(* IEC 61131-3 sources: mect_apps/AnyTPAC/TestSuite/plc (part 2) *)

(* ---- eq_P.st ---- *)
(*[[
]]*)
PROGRAM eq_P
#import "Crosstable.gvl"
#import "Resource1.gvl"
CONST
	this : int := 36;
	test_cases : int := 6;
END_CONST
VAR
	test_case : array [1..test_cases] of any2_bool_T := [
		(input0 :=  10.0, input1 :=  10.0, retval := true),
		(input0 :=  10.0, input1 :=  20.0, retval := false),
		(input0 :=  10.0, input1 :=  5.0,  retval := false),
		(input0 :=  -100.0, input1 := -100.0,  retval := true),
		(input0 :=  -100.0, input1 := 7.0,  retval := false),
		(input0 :=  -100.0, input1 := 109.0,  retval := false)
	];
	ret_bool   : bool;
	ret_byte   : bool;
	ret_dint   : bool;
	ret_dword  : bool;
	ret_int    : bool;
	ret_lreal  : bool;
	ret_real   : bool;
	ret_string : bool;
	ret_time   : bool;
	ret_uint   : bool;
	ret_udint  : bool;
	ret_word   : bool;

	expected_ret_bool   : bool;
	expected_ret_byte   : bool;
	expected_ret_dint   : bool;
	expected_ret_dword  : bool;
	expected_ret_int    : bool;
	expected_ret_lreal  : bool;
	expected_ret_real   : bool;
	expected_ret_string : bool;
	expected_ret_time   : bool;
	expected_ret_uint   : bool;
	expected_ret_udint  : bool;
	expected_ret_word   : bool;

	index : int := 1;
	expected: string;
	obtained: string;
	result : bool;
END_VAR

	if Status = STATUS_RUNNING AND test_level_36 > TEST_DISABLED and test_loops_36 < Target then

		(* ---------- test action ---------------*)
        ret_bool   := eq( lreal_to_bool(test_case[index].input0),
						 lreal_to_bool(test_case[index].input1));
        ret_byte   := eq( lreal_to_byte(test_case[index].input0),
						 lreal_to_byte(test_case[index].input1));
        ret_dint   := eq( lreal_to_dint(test_case[index].input0),
						 lreal_to_dint(test_case[index].input1));
        ret_dword  := eq( lreal_to_dword(test_case[index].input0),
						 lreal_to_dword(test_case[index].input1));
        ret_int    := eq( lreal_to_int(test_case[index].input0),
						 lreal_to_int(test_case[index].input1));
        ret_lreal  := eq( test_case[index].input0,
						 test_case[index].input1);
        ret_real   := eq( lreal_to_real(test_case[index].input0),
						 lreal_to_real(test_case[index].input1));
        ret_string := eq(lreal_to_string(test_case[index].input0),
						 lreal_to_string(test_case[index].input1));
        ret_time   := eq( lreal_to_time(test_case[index].input0),
						 lreal_to_time(test_case[index].input1));
        ret_uint   := eq( lreal_to_uint(test_case[index].input0),
						 lreal_to_uint(test_case[index].input1));
        ret_udint  := eq(lreal_to_udint(test_case[index].input0),
						 lreal_to_udint(test_case[index].input1));
        ret_word   := eq( lreal_to_word(test_case[index].input0),
						 lreal_to_word(test_case[index].input1));

		IF (test_case[index].input0 <> 0.0 and test_case[index].input1 <> 0.0)
			or (test_case[index].input0 = 0.0 and test_case[index].input1 = 0.0)THEN
        	expected_ret_bool   := true;
        ELSE
        	expected_ret_bool   := false;
		END_IF;

		expected_ret_byte   := test_case[index].retval;
		expected_ret_dint   := test_case[index].retval;
		expected_ret_dword  := test_case[index].retval;
		expected_ret_int    := test_case[index].retval;
		expected_ret_lreal  := test_case[index].retval;
		expected_ret_real   := test_case[index].retval;
		expected_ret_string := test_case[index].retval;
		expected_ret_time   := test_case[index].retval;
		expected_ret_uint   := test_case[index].retval;
		expected_ret_udint  := test_case[index].retval;
		expected_ret_word   := test_case[index].retval;

		(* ---------- test condition ---------------*)
        result := (ret_bool = expected_ret_bool)
				  and (ret_byte = expected_ret_byte)
				  and (ret_dint = expected_ret_dint)
				  and (ret_dword = expected_ret_dword)
				  and (ret_int = expected_ret_int)
				  and (ret_lreal = expected_ret_lreal)
				  and (ret_real = expected_ret_real)
				  and (ret_string = expected_ret_string)
				  and (ret_time = expected_ret_time)
				  and (ret_uint = expected_ret_uint)
				  and (ret_udint = expected_ret_udint)
				  and (ret_word = expected_ret_word);

		(* ---------- log message ---------------*)
		expected := '';
		expected := CONCAT(expected, comma_blank, bool_to_string(expected_ret_bool));
		expected := CONCAT(expected, comma_blank, bool_to_string(expected_ret_byte));
		expected := CONCAT(expected, comma_blank, bool_to_string(expected_ret_dint));
		expected := CONCAT(expected, comma_blank, bool_to_string(expected_ret_dword));
		expected := CONCAT(expected, comma_blank, bool_to_string(expected_ret_int));
		expected := CONCAT(expected, comma_blank, bool_to_string(expected_ret_lreal));
		expected := CONCAT(expected, comma_blank, bool_to_string(expected_ret_real));
		expected := CONCAT(expected, comma_blank, bool_to_string(expected_ret_string));
		expected := CONCAT(expected, comma_blank, bool_to_string(expected_ret_time));
		expected := CONCAT(expected, comma_blank, bool_to_string(expected_ret_uint));
		expected := CONCAT(expected, comma_blank, bool_to_string(expected_ret_udint));
		expected := CONCAT(expected, comma_blank, bool_to_string(expected_ret_word));

		obtained := '';
		obtained := CONCAT(obtained, comma_blank, bool_to_string(ret_bool));
		obtained := CONCAT(obtained, comma_blank, bool_to_string(ret_byte));
		obtained := CONCAT(obtained, comma_blank, bool_to_string(ret_dint));
		obtained := CONCAT(obtained, comma_blank, bool_to_string(ret_dword));
		obtained := CONCAT(obtained, comma_blank, bool_to_string(ret_int));
		obtained := CONCAT(obtained, comma_blank, bool_to_string(ret_lreal));
		obtained := CONCAT(obtained, comma_blank, bool_to_string(ret_real));
		obtained := CONCAT(obtained, comma_blank, bool_to_string(ret_string));
		obtained := CONCAT(obtained, comma_blank, bool_to_string(ret_time));
		obtained := CONCAT(obtained, comma_blank, bool_to_string(ret_uint));
		obtained := CONCAT(obtained, comma_blank, bool_to_string(ret_udint));
		obtained := CONCAT(obtained, comma_blank, bool_to_string(ret_word));

		(* ---------- cycle ----------*)
		SingleTest(this, result, expected, obtained, test_cases,
				   index, test_level_36, test_counter_36, test_loops_36, test_errors_36);
	end_if;

END_PROGRAM

(* ---- expt_P.st ---- *)
(*[[ ]]*)
PROGRAM expt_P
#import "Crosstable.gvl"
#import "Resource1.gvl"
CONST
	this : int := 20;
	test_cases : int := 5;
	xl : lreal := 0.0000000000001;
	x : real := 0.0000000000001;
END_CONST
VAR
	test_case : array [1..test_cases] of num2_num_T := [
		(input0 := 2.0, input1 := 2.0, ret_real := 4.0, ret_lreal := 4.0),
		(input0 := 2.0, input1 := 3.0, ret_real := 8.0, ret_lreal := 8.0),
		(input0 := 10.0, input1 := 2.0, ret_real := 100.0, ret_lreal := 100.0),
		(input0 := 5.0, input1 := 3.0, ret_real := 125.0, ret_lreal := 125.0),
		(input0 := 10.0, input1 := -1.0, ret_real := 0.1, ret_lreal := 0.1)
	];
    ret_real_int    : real;
    ret_real_dint   : real;
    ret_real_real   : real;
    ret_real_lreal  : real;
    ret_lreal_int   : lreal;
    ret_lreal_dint  : lreal;
    ret_lreal_real  : lreal;
    ret_lreal_lreal : lreal;

	index : int := 1;
	expected : string;
	obtained : string;
	result : bool;
END_VAR

	if Status = STATUS_RUNNING AND test_level_20 > TEST_DISABLED and test_loops_20 < Target then

		(* ---------- test action ---------------*)
        ret_real_int   := expt(lreal_to_real(test_case[index].input0), lreal_to_int(test_case[index].input1));
        ret_real_dint  := expt(lreal_to_real(test_case[index].input0), lreal_to_dint(test_case[index].input1));
        ret_real_real  := expt(lreal_to_real(test_case[index].input0), lreal_to_real(test_case[index].input1));
        ret_real_lreal := expt(lreal_to_real(test_case[index].input0), test_case[index].input1);

        ret_lreal_int   := expt(test_case[index].input0, lreal_to_int(test_case[index].input1));
        ret_lreal_dint  := expt(test_case[index].input0, lreal_to_dint(test_case[index].input1));
        ret_lreal_real  := expt(test_case[index].input0, lreal_to_real(test_case[index].input1));
        ret_lreal_lreal := expt(test_case[index].input0, test_case[index].input1);

		(* ---------- test condition ---------------*)
        result := ((abs(ret_real_int - test_case[index].ret_real) < x)
		      and (abs(ret_real_dint - test_case[index].ret_real) < x)
		      and (abs(ret_real_real - test_case[index].ret_real) < x)
		      and (abs(ret_real_lreal - test_case[index].ret_real) < x)
			  and (abs(ret_lreal_int - test_case[index].ret_lreal) < xl)
		      and (abs(ret_lreal_dint - test_case[index].ret_lreal) < xl)
		      and (abs(ret_lreal_real - test_case[index].ret_lreal) < xl)
		      and (abs(ret_lreal_lreal - test_case[index].ret_lreal) < xl));

		(* ---------- log message ---------------*)
		expected := '';
		expected := CONCAT(expected, comma_blank, real_to_string(test_case[index].ret_real));
		expected := CONCAT(expected, comma_blank, real_to_string(test_case[index].ret_real));
		expected := CONCAT(expected, comma_blank, real_to_string(test_case[index].ret_real));
		expected := CONCAT(expected, comma_blank, real_to_string(test_case[index].ret_real));
		expected := CONCAT(expected, comma_blank, lreal_to_string(test_case[index].ret_lreal));
		expected := CONCAT(expected, comma_blank, lreal_to_string(test_case[index].ret_lreal));
		expected := CONCAT(expected, comma_blank, lreal_to_string(test_case[index].ret_lreal));
		expected := CONCAT(expected, comma_blank, lreal_to_string(test_case[index].ret_lreal));
		obtained := '';
		obtained := CONCAT(obtained, comma_blank, real_to_string(ret_real_int));
		obtained := CONCAT(obtained, comma_blank, real_to_string(ret_real_dint));
		obtained := CONCAT(obtained, comma_blank, real_to_string(ret_real_real));
		obtained := CONCAT(obtained, comma_blank, real_to_string(ret_real_lreal));
		obtained := CONCAT(obtained, comma_blank, lreal_to_string(ret_lreal_int));
		obtained := CONCAT(obtained, comma_blank, lreal_to_string(ret_lreal_dint));
		obtained := CONCAT(obtained, comma_blank, lreal_to_string(ret_lreal_real));
		obtained := CONCAT(obtained, comma_blank, lreal_to_string(ret_lreal_lreal));

		(* ---------- cycle ----------*)
		SingleTest(this, result, expected, obtained, test_cases,
				   index, test_level_20, test_counter_20, test_loops_20, test_errors_20);
	end_if;
END_PROGRAM

(* ---- f_r_trig_P.st ---- *)
(*[[
]]*)
PROGRAM f_r_trig_P
#import "Crosstable.gvl"
#import "Resource1.gvl"
CONST
	this : int := 53;
	test_cases : int := 5;
END_CONST
VAR
	test_case : array [1..test_cases] of bool_bool2_T := [
		(input := false, retval1 := false, retval2 := false),
		(input := true,  retval1 := false, retval2 := true ),
		(input := true,  retval1 := false, retval2 := false),
		(input := false, retval1 := true,  retval2 := false),
		(input := false, retval1 := false, retval2 := false)
	];
    retval1  : bool;
    retval2  : bool;

	F_TRIG_Inst : f_trig;
	R_TRIG_Inst : r_trig;
	index : int := 1;
	expected : string;
	obtained : string;
	result : bool;
END_VAR

	if Status = STATUS_RUNNING AND test_level_53 > TEST_DISABLED and test_loops_53 < Target then

		(* ---------- test action ---------------*)
		F_TRIG_Inst(CLK := test_case[index].input, Q => retval1);
		R_TRIG_Inst(CLK := test_case[index].input, Q => retval2);

		(* ---------- test condition ---------------*)
        result := (retval1 = test_case[index].retval1)
		      and (retval2 = test_case[index].retval2);

		(* ---------- log message ---------------*)
		expected := '';
		expected := CONCAT(expected, comma_blank, bool_to_string(test_case[index].retval1));
		expected := CONCAT(expected, comma_blank, bool_to_string(test_case[index].retval2));
		obtained := '';
		obtained := CONCAT(obtained, comma_blank, bool_to_string(retval1));
		obtained := CONCAT(obtained, comma_blank, bool_to_string(retval2));

		(* ---------- cycle ----------*)
		SingleTest(this, result, expected, obtained, test_cases,
				   index, test_level_53, test_counter_53, test_loops_53, test_errors_53);
	end_if;
END_PROGRAM

(* ---- find_P.st ---- *)
(*[[ ]]*)
PROGRAM find_P
#import "Crosstable.gvl"
#import "Resource1.gvl"
CONST
	this : int := 44;
	test_cases : int := 4;
END_CONST
VAR
	test_case : array [1..test_cases] of string2_int_T := [
		(input0 := 'stringa_in_cui_eseguire_la_ricerca', input1 := 'stringa',  retval := 1),
		(input0 := 'stringa_in_cui_eseguire_la_ricerca', input1 := 'in_cui',   retval := 9),
		(input0 := 'stringa_in_cui_eseguire_la_ricerca', input1 := 'ricerca',  retval := 28),
		(input0 := 'stringa_in_cui_eseguire_la_ricerca', input1 := 'stringa_che_non_esiste',  retval := 0)
	];
    retval0   : int;
    retval1   : dint;

	index : int := 1;
	expected : string;
	obtained : string;
	result : bool;
END_VAR

	if Status = STATUS_RUNNING AND test_level_44 > TEST_DISABLED and test_loops_44 < Target then

		(* ---------- test action ---------------*)
        retval0 := find(test_case[index].input0, test_case[index].input1);
        retval1 := find(test_case[index].input0, test_case[index].input1);

		(* ---------- test condition ---------------*)
        result := (retval0 = test_case[index].retval)
		      and (retval1 = int_to_dint(test_case[index].retval));

		(* ---------- log message ---------------*)
		expected := '';
		expected := CONCAT(expected, comma_blank, int_to_string(test_case[index].retval));
		expected := CONCAT(expected, comma_blank, int_to_string(test_case[index].retval));
		obtained := '';
		obtained := CONCAT(obtained, comma_blank, int_to_string(retval0));
		obtained := CONCAT(obtained, comma_blank, dint_to_string(retval1));

		(* ---------- cycle ----------*)
		SingleTest(this, result, expected, obtained, test_cases,
				   index, test_level_44, test_counter_44, test_loops_44, test_errors_44);
	end_if;
END_PROGRAM

(* ---- ge_P.st ---- *)
(*[[
]]*)
PROGRAM ge_P
#import "Crosstable.gvl"
#import "Resource1.gvl"
CONST
	this : int := 37;
	test_cases : int := 4;
END_CONST
VAR
	test_case : array [1..test_cases] of any2_bool_T := [
		(input0 :=  10.0, input1 :=  10.0, retval := true),
		(input0 :=  10.0, input1 :=  20.0, retval := false),
		(input0 :=  20.0, input1 :=  10.0,  retval := true),
		(input0 :=  -100.0, input1 := -100.0,  retval := true)
	];
	ret_bool   : bool;
	ret_byte   : bool;
	ret_dint   : bool;
	ret_dword  : bool;
	ret_int    : bool;
	ret_lreal  : bool;
	ret_real   : bool;
	ret_string : bool;
	ret_time   : bool;
	ret_uint   : bool;
	ret_udint  : bool;
	ret_word   : bool;

	expected_ret_bool   : bool;
	expected_ret_byte   : bool;
	expected_ret_dint   : bool;
	expected_ret_dword  : bool;
	expected_ret_int    : bool;
	expected_ret_lreal  : bool;
	expected_ret_real   : bool;
	expected_ret_string : bool;
	expected_ret_time   : bool;
	expected_ret_uint   : bool;
	expected_ret_udint  : bool;
	expected_ret_word   : bool;

	index : int := 1;
	expected: string;
	obtained: string;
	result : bool;
END_VAR

	if Status = STATUS_RUNNING AND test_level_37 > TEST_DISABLED and test_loops_37 < Target then

		(* ---------- test action ---------------*)
        ret_bool   := ge( lreal_to_bool(test_case[index].input0),
						 lreal_to_bool(test_case[index].input1));
        ret_byte   := ge( lreal_to_byte(test_case[index].input0),
						 lreal_to_byte(test_case[index].input1));
        ret_dint   := ge( lreal_to_dint(test_case[index].input0),
						 lreal_to_dint(test_case[index].input1));
        ret_dword  := ge( lreal_to_dword(test_case[index].input0),
						 lreal_to_dword(test_case[index].input1));
        ret_int    := ge( lreal_to_int(test_case[index].input0),
						 lreal_to_int(test_case[index].input1));
        ret_lreal  := ge( test_case[index].input0,
						 test_case[index].input1);
        ret_real   := ge( lreal_to_real(test_case[index].input0),
						 lreal_to_real(test_case[index].input1));
        ret_string := ge(lreal_to_string(test_case[index].input0),
						 lreal_to_string(test_case[index].input1));
        ret_time   := ge( lreal_to_time(test_case[index].input0),
						 lreal_to_time(test_case[index].input1));
        ret_uint   := ge( lreal_to_uint(test_case[index].input0),
						 lreal_to_uint(test_case[index].input1));
        ret_udint  := ge(lreal_to_udint(test_case[index].input0),
						 lreal_to_udint(test_case[index].input1));
        ret_word   := ge( lreal_to_word(test_case[index].input0),
						 lreal_to_word(test_case[index].input1));

		IF (test_case[index].input0 <> 0.0 and test_case[index].input1 <> 0.0)
			or (test_case[index].input0 = 0.0 and test_case[index].input1 = 0.0)THEN
        	expected_ret_bool   := true;
        ELSE
        	expected_ret_bool   := false;
		END_IF;
		expected_ret_byte   := test_case[index].retval;
		expected_ret_dint   := test_case[index].retval;
		expected_ret_dword  := test_case[index].retval;
		expected_ret_int    := test_case[index].retval;
		expected_ret_lreal  := test_case[index].retval;
		expected_ret_real   := test_case[index].retval;
		expected_ret_string := test_case[index].retval;
		expected_ret_time   := test_case[index].retval;
		expected_ret_uint   := test_case[index].retval;
		expected_ret_udint  := test_case[index].retval;
		expected_ret_word   := test_case[index].retval;

		(* ---------- test condition ---------------*)
        result := (ret_bool = expected_ret_bool)
				  and (ret_byte = expected_ret_byte)
				  and (ret_dint = expected_ret_dint)
				  and (ret_dword = expected_ret_dword)
				  and (ret_int = expected_ret_int)
				  and (ret_lreal = expected_ret_lreal)
				  and (ret_real = expected_ret_real)
				  and (ret_string = expected_ret_string)
				  and (ret_time = expected_ret_time)
				  and (ret_uint = expected_ret_uint)
				  and (ret_udint = expected_ret_udint)
				  and (ret_word = expected_ret_word);

		(* ---------- log message ---------------*)
		expected := '';
		expected := CONCAT(expected, comma_blank, bool_to_string(expected_ret_bool));
		expected := CONCAT(expected, comma_blank, bool_to_string(expected_ret_byte));
		expected := CONCAT(expected, comma_blank, bool_to_string(expected_ret_dint));
		expected := CONCAT(expected, comma_blank, bool_to_string(expected_ret_dword));
		expected := CONCAT(expected, comma_blank, bool_to_string(expected_ret_int));
		expected := CONCAT(expected, comma_blank, bool_to_string(expected_ret_lreal));
		expected := CONCAT(expected, comma_blank, bool_to_string(expected_ret_real));
		expected := CONCAT(expected, comma_blank, bool_to_string(expected_ret_string));
		expected := CONCAT(expected, comma_blank, bool_to_string(expected_ret_time));
		expected := CONCAT(expected, comma_blank, bool_to_string(expected_ret_uint));
		expected := CONCAT(expected, comma_blank, bool_to_string(expected_ret_udint));
		expected := CONCAT(expected, comma_blank, bool_to_string(expected_ret_word));

		obtained := '';
		obtained := CONCAT(obtained, comma_blank, bool_to_string(ret_bool));
		obtained := CONCAT(obtained, comma_blank, bool_to_string(ret_byte));
		obtained := CONCAT(obtained, comma_blank, bool_to_string(ret_dint));
		obtained := CONCAT(obtained, comma_blank, bool_to_string(ret_dword));
		obtained := CONCAT(obtained, comma_blank, bool_to_string(ret_int));
		obtained := CONCAT(obtained, comma_blank, bool_to_string(ret_lreal));
		obtained := CONCAT(obtained, comma_blank, bool_to_string(ret_real));
		obtained := CONCAT(obtained, comma_blank, bool_to_string(ret_string));
		obtained := CONCAT(obtained, comma_blank, bool_to_string(ret_time));
		obtained := CONCAT(obtained, comma_blank, bool_to_string(ret_uint));
		obtained := CONCAT(obtained, comma_blank, bool_to_string(ret_udint));
		obtained := CONCAT(obtained, comma_blank, bool_to_string(ret_word));

		(* ---------- cycle ----------*)
		SingleTest(this, result, expected, obtained, test_cases,
				   index, test_level_37, test_counter_37, test_loops_37, test_errors_37);
	end_if;

END_PROGRAM

(* ---- gt_P.st ---- *)
(*[[
]]*)
PROGRAM gt_P
#import "Crosstable.gvl"
#import "Resource1.gvl"
CONST
	this : int := 38;
	test_cases : int := 4;
END_CONST
VAR
	test_case : array [1..test_cases] of any2_bool_T := [
		(input0 :=  10.0, input1 :=  10.0, retval := false),
		(input0 :=  10.0, input1 :=  20.0, retval := false),
		(input0 :=  20.0, input1 :=  10.0,  retval := true),
		(input0 :=  -100.0, input1 := -100.0,  retval := false)
	];
	ret_bool   : bool;
	ret_byte   : bool;
	ret_dint   : bool;
	ret_dword  : bool;
	ret_int    : bool;
	ret_lreal  : bool;
	ret_real   : bool;
	ret_string : bool;
	ret_time   : bool;
	ret_uint   : bool;
	ret_udint  : bool;
	ret_word   : bool;

	expected_ret_bool   : bool;
	expected_ret_byte   : bool;
	expected_ret_dint   : bool;
	expected_ret_dword  : bool;
	expected_ret_int    : bool;
	expected_ret_lreal  : bool;
	expected_ret_real   : bool;
	expected_ret_string : bool;
	expected_ret_time   : bool;
	expected_ret_uint   : bool;
	expected_ret_udint  : bool;
	expected_ret_word   : bool;

	index : int := 1;
	expected: string;
	obtained: string;
	result : bool;
END_VAR

	if Status = STATUS_RUNNING AND test_level_38 > TEST_DISABLED and test_loops_38 < Target then

		(* ---------- test action ---------------*)
        ret_bool   := gt( lreal_to_bool(test_case[index].input0),
						 lreal_to_bool(test_case[index].input1));
        ret_byte   := gt( lreal_to_byte(test_case[index].input0),
						 lreal_to_byte(test_case[index].input1));
        ret_dint   := gt( lreal_to_dint(test_case[index].input0),
						 lreal_to_dint(test_case[index].input1));
        ret_dword  := gt( lreal_to_dword(test_case[index].input0),
						 lreal_to_dword(test_case[index].input1));
        ret_int    := gt( lreal_to_int(test_case[index].input0),
						 lreal_to_int(test_case[index].input1));
        ret_lreal  := gt( test_case[index].input0,
						 test_case[index].input1);
        ret_real   := gt( lreal_to_real(test_case[index].input0),
						 lreal_to_real(test_case[index].input1));
        ret_string := gt(lreal_to_string(test_case[index].input0),
						 lreal_to_string(test_case[index].input1));
        ret_time   := gt( lreal_to_time(test_case[index].input0),
						 lreal_to_time(test_case[index].input1));
        ret_uint   := gt( lreal_to_uint(test_case[index].input0),
						 lreal_to_uint(test_case[index].input1));
        ret_udint  := gt(lreal_to_udint(test_case[index].input0),
						 lreal_to_udint(test_case[index].input1));
        ret_word   := gt( lreal_to_word(test_case[index].input0),
						 lreal_to_word(test_case[index].input1));

		IF (test_case[index].input0 <> 0.0 and test_case[index].input1 <> 0.0)
			or (test_case[index].input0 = 0.0 and test_case[index].input1 = 0.0)THEN
        	expected_ret_bool   := false;
        ELSE
        	expected_ret_bool   := true;
		END_IF;
		expected_ret_byte   := test_case[index].retval;
		expected_ret_dint   := test_case[index].retval;
		expected_ret_dword  := test_case[index].retval;
		expected_ret_int    := test_case[index].retval;
		expected_ret_lreal  := test_case[index].retval;
		expected_ret_real   := test_case[index].retval;
		expected_ret_string := test_case[index].retval;
		expected_ret_time   := test_case[index].retval;
		expected_ret_uint   := test_case[index].retval;
		expected_ret_udint  := test_case[index].retval;
		expected_ret_word   := test_case[index].retval;

		(* ---------- test condition ---------------*)
        result := (ret_bool = expected_ret_bool)
				  and (ret_byte = expected_ret_byte)
				  and (ret_dint = expected_ret_dint)
				  and (ret_dword = expected_ret_dword)
				  and (ret_int = expected_ret_int)
				  and (ret_lreal = expected_ret_lreal)
				  and (ret_real = expected_ret_real)
				  and (ret_string = expected_ret_string)
				  and (ret_time = expected_ret_time)
				  and (ret_uint = expected_ret_uint)
				  and (ret_udint = expected_ret_udint)
				  and (ret_word = expected_ret_word);

		(* ---------- log message ---------------*)
		expected := '';
		expected := CONCAT(expected, comma_blank, bool_to_string(expected_ret_bool));
		expected := CONCAT(expected, comma_blank, bool_to_string(expected_ret_byte));
		expected := CONCAT(expected, comma_blank, bool_to_string(expected_ret_dint));
		expected := CONCAT(expected, comma_blank, bool_to_string(expected_ret_dword));
		expected := CONCAT(expected, comma_blank, bool_to_string(expected_ret_int));
		expected := CONCAT(expected, comma_blank, bool_to_string(expected_ret_lreal));
		expected := CONCAT(expected, comma_blank, bool_to_string(expected_ret_real));
		expected := CONCAT(expected, comma_blank, bool_to_string(expected_ret_string));
		expected := CONCAT(expected, comma_blank, bool_to_string(expected_ret_time));
		expected := CONCAT(expected, comma_blank, bool_to_string(expected_ret_uint));
		expected := CONCAT(expected, comma_blank, bool_to_string(expected_ret_udint));
		expected := CONCAT(expected, comma_blank, bool_to_string(expected_ret_word));

		obtained := '';
		obtained := CONCAT(obtained, comma_blank, bool_to_string(ret_bool));
		obtained := CONCAT(obtained, comma_blank, bool_to_string(ret_byte));
		obtained := CONCAT(obtained, comma_blank, bool_to_string(ret_dint));
		obtained := CONCAT(obtained, comma_blank, bool_to_string(ret_dword));
		obtained := CONCAT(obtained, comma_blank, bool_to_string(ret_int));
		obtained := CONCAT(obtained, comma_blank, bool_to_string(ret_lreal));
		obtained := CONCAT(obtained, comma_blank, bool_to_string(ret_real));
		obtained := CONCAT(obtained, comma_blank, bool_to_string(ret_string));
		obtained := CONCAT(obtained, comma_blank, bool_to_string(ret_time));
		obtained := CONCAT(obtained, comma_blank, bool_to_string(ret_uint));
		obtained := CONCAT(obtained, comma_blank, bool_to_string(ret_udint));
		obtained := CONCAT(obtained, comma_blank, bool_to_string(ret_word));

		(* ---------- cycle ----------*)
		SingleTest(this, result, expected, obtained, test_cases,
				   index, test_level_38, test_counter_38, test_loops_38, test_errors_38);
	end_if;

END_PROGRAM

(* ---- hi_byte_P.st ---- *)
(*[[
]]*)
PROGRAM hi_byte_P
#import "Crosstable.gvl"
#import "Resource1.gvl"
CONST
	this : int := 58;
	test_cases : int := 4;
END_CONST
VAR
	test_case : array [1..test_cases] of bit_bit2_T := [
		(input := 0, 			ret_byte := 16#00, ret_word := 16#0000, ret_byte2 := 16#00, ret_word2 := 16#0000),
		(input := 16#ffffffff, 	ret_byte := 16#ff, ret_word := 16#ffff, ret_byte2 := 16#ff, ret_word2 := 16#ffff),
		(input := 16#5678, 		ret_byte := 16#56, ret_word := 16#0000, ret_byte2 := 16#78, ret_word2 := 16#5678),
		(input := 16#12345678, 	ret_byte := 16#56, ret_word := 16#1234, ret_byte2 := 16#78, ret_word2 := 16#5678)
	];
    ret_byte   : byte;
    ret_word   : word;
    ret_byte2  : byte;
    ret_word2  : word;

	index : int := 1;
	expected : string;
	obtained : string;
	result : bool;
END_VAR

	if Status = STATUS_RUNNING AND test_level_58 > TEST_DISABLED and test_loops_58 < Target then

		(* ---------- test action ---------------*)
        ret_byte   := hi_byte(dword_to_word(test_case[index].input));
        ret_word   := hi_word(test_case[index].input);
        ret_byte2  := lo_byte(dword_to_word(test_case[index].input));
        ret_word2  := lo_word(test_case[index].input);

		(* ---------- test condition ---------------*)
        result := (ret_byte = test_case[index].ret_byte)
			  and (ret_word = test_case[index].ret_word)
			  and (ret_byte2 = test_case[index].ret_byte2)
			  and (ret_word2 = test_case[index].ret_word2);

		(* ---------- log message ---------------*)
		expected := '';
		expected := CONCAT(expected, comma_blank, byte_to_string(test_case[index].ret_byte));
		expected := CONCAT(expected, comma_blank, word_to_string(test_case[index].ret_word));
		expected := CONCAT(expected, comma_blank, byte_to_string(test_case[index].ret_byte2));
		expected := CONCAT(expected, comma_blank, word_to_string(test_case[index].ret_word2));
		obtained := '';
		obtained := CONCAT(obtained, comma_blank, byte_to_string(ret_byte));
		obtained := CONCAT(obtained, comma_blank, word_to_string(ret_word));
		obtained := CONCAT(obtained, comma_blank, byte_to_string(ret_byte2));
		obtained := CONCAT(obtained, comma_blank, word_to_string(ret_word2));

		(* ---------- cycle ----------*)
		SingleTest(this, result, expected, obtained, test_cases,
				   index, test_level_58, test_counter_58, test_loops_58, test_errors_58);
	end_if;
END_PROGRAM

(* ---- insert_P.st ---- *)
(*[[ ]]*)
PROGRAM insert_P
#import "Crosstable.gvl"
#import "Resource1.gvl"
CONST
	this : int := 45;
	test_cases : int := 3;
END_CONST
VAR
	test_case : array [1..test_cases] of string2_int_string_T := [
		(input0 := 'stringa_dove_inserire', input1 := 'abc_', input2 := 0,  retval := 'abc_stringa_dove_inserire'),
		(input0 := 'stringa_dove_inserire', input1 := 'abc_', input2 := 8,  retval := 'stringa_abc_dove_inserire'),
		(input0 := 'stringa_dove_inserire', input1 := 'abc_', input2 := 21, retval := 'stringa_dove_inserireabc_')
	];
    retval0   : string;
    retval1   : string;

	index : int := 1;
	expected : string;
	obtained : string;
	result : bool;
END_VAR

	if Status = STATUS_RUNNING AND test_level_45 > TEST_DISABLED and test_loops_45 < Target then

		(* ---------- test action ---------------*)
        retval0 := insert(test_case[index].input0, test_case[index].input1, test_case[index].input2);
        retval1 := insert(test_case[index].input0, test_case[index].input1, int_to_dint(test_case[index].input2));

		(* ---------- test condition ---------------*)
        result := (retval0 = test_case[index].retval)
		      and (retval1 = test_case[index].retval);

		(* ---------- log message ---------------*)
		expected := '';
		expected := CONCAT(expected, comma_blank, test_case[index].retval);
		expected := CONCAT(expected, comma_blank, test_case[index].retval);
		obtained := '';
		obtained := CONCAT(obtained, comma_blank, retval0);
		obtained := CONCAT(obtained, comma_blank, retval1);

		(* ---------- cycle ----------*)
		SingleTest(this, result, expected, obtained, test_cases,
				   index, test_level_45, test_counter_45, test_loops_45, test_errors_45);
	end_if;
END_PROGRAM

(* ---- int_to_all_P.st ---- *)
(*[[
]]*)
PROGRAM int_to_all_P
#import "Crosstable.gvl"
#import "Resource1.gvl"
CONST
	this : int := 5;
	test_cases : int := 4;
END_CONST
VAR
	test_case : array [1..test_cases] of dword_all_T := [
		(input := 0, ret_bool := 0, ret_byte := 0, ret_dint := 0, ret_int := 0, ret_lreal := 0.0, ret_real := 0.0,
		   ret_string := '0', ret_udint := 0, ret_uint := 0, ret_word := 0),
		(input := 1, ret_bool := 1, ret_byte := 1, ret_dint := 1, ret_int := 1, ret_lreal := 1.0, ret_real := 1.0,
		   ret_string := '1', ret_udint := 1, ret_uint := 1, ret_word := 1),
		(input := 255, ret_bool := 1, ret_byte := 255, ret_dint := 255, ret_int := 255, ret_lreal := 255.0, ret_real := 255.0,
		   ret_string := '255', ret_udint := 255, ret_uint := 255, ret_word := 255),
		(input := 400, ret_bool := 1, ret_byte := 144, ret_dint := 400, ret_int := 400, ret_lreal := 400.0, ret_real := 400.0,
		   ret_string := '400', ret_udint := 400, ret_uint := 400, ret_word := 400)
	];
    ret_bool   : bool;
    ret_byte   : byte;
    ret_dint   : dint;
    ret_int    : int;
    ret_lreal  : lreal;
    ret_real   : real;
    ret_string : string;
    ret_udint  : udint;
    ret_uint   : uint;
    ret_word   : word;

	index : int := 1;
	expected : string;
	obtained : string;
	result : bool;
END_VAR

	if Status = STATUS_RUNNING AND test_level_05 > TEST_DISABLED and test_loops_05 < Target then

		(* ---------- test action ---------------*)
        ret_bool   := dword_to_bool(test_case[index].input);
        ret_byte   := dword_to_byte(test_case[index].input);
        ret_dint   := dword_to_dint(test_case[index].input);
        ret_int    := dword_to_int(test_case[index].input);
        ret_lreal  := dword_to_lreal(test_case[index].input);
        ret_real   := dword_to_real(test_case[index].input);
        ret_string := dword_to_string(test_case[index].input);
        ret_udint  := dword_to_udint(test_case[index].input);
        ret_uint   := dword_to_uint(test_case[index].input);
        ret_word   := dword_to_word(test_case[index].input);

		(* ---------- test condition ---------------*)
        result := (ret_bool = test_case[index].ret_bool)
		      and (ret_byte = test_case[index].ret_byte)
		      and (ret_dint = test_case[index].ret_dint)
		      and (ret_int = test_case[index].ret_int)
		      and (ret_lreal = test_case[index].ret_lreal)
		      and (ret_real = test_case[index].ret_real)
		      and (ret_string = test_case[index].ret_string)
		      and (ret_udint = test_case[index].ret_udint)
		      and (ret_uint = test_case[index].ret_uint)
		      and (ret_word = test_case[index].ret_word);

		(* ---------- log message ---------------*)
		expected := '';
		expected := CONCAT(expected, comma_blank, bool_to_string(test_case[index].ret_bool));
		expected := CONCAT(expected, comma_blank, byte_to_string(test_case[index].ret_byte));
		expected := CONCAT(expected, comma_blank, dint_to_string(test_case[index].ret_dint));
		expected := CONCAT(expected, comma_blank, int_to_string(test_case[index].ret_int));
		expected := CONCAT(expected, comma_blank, lreal_to_string(test_case[index].ret_lreal));
		expected := CONCAT(expected, comma_blank, real_to_string(test_case[index].ret_real));
		expected := CONCAT(expected, comma_blank, test_case[index].ret_string);
		expected := CONCAT(expected, comma_blank, udint_to_string(test_case[index].ret_udint));
		expected := CONCAT(expected, comma_blank, uint_to_string(test_case[index].ret_uint));
		expected := CONCAT(expected, comma_blank, word_to_string(test_case[index].ret_word));
		obtained := '';
		obtained := CONCAT(obtained, comma_blank, bool_to_string(ret_bool));
		obtained := CONCAT(obtained, comma_blank, byte_to_string(ret_byte));
		obtained := CONCAT(obtained, comma_blank, dint_to_string(ret_dint));
		obtained := CONCAT(obtained, comma_blank, int_to_string(ret_int));
		obtained := CONCAT(obtained, comma_blank, lreal_to_string(ret_lreal));
		obtained := CONCAT(obtained, comma_blank, real_to_string(ret_real));
		obtained := CONCAT(obtained, comma_blank, ret_string);
		obtained := CONCAT(obtained, comma_blank, udint_to_string(ret_udint));
		obtained := CONCAT(obtained, comma_blank, uint_to_string(ret_uint));
		obtained := CONCAT(obtained, comma_blank, word_to_string(ret_word));

		(* ---------- cycle ----------*)
		SingleTest(this, result, expected, obtained, test_cases,
				   index, test_level_05, test_counter_05, test_loops_05, test_errors_05);
	end_if;

END_PROGRAM

(* ---- le_P.st ---- *)
(*[[
]]*)
PROGRAM le_P
#import "Crosstable.gvl"
#import "Resource1.gvl"
CONST
	this : int := 39;
	test_cases : int := 4;
END_CONST
VAR
	test_case : array [1..test_cases] of any2_bool_T := [
		(input0 :=  10.0, input1 :=  10.0, retval := true),
		(input0 :=  10.0, input1 :=  20.0, retval := true),
		(input0 :=  20.0, input1 :=  10.0,  retval := false),
		(input0 :=  -100.0, input1 := -100.0,  retval := true)
	];
	ret_bool   : bool;
	ret_byte   : bool;
	ret_dint   : bool;
	ret_dword  : bool;
	ret_int    : bool;
	ret_lreal  : bool;
	ret_real   : bool;
	ret_string : bool;
	ret_time   : bool;
	ret_uint   : bool;
	ret_udint  : bool;
	ret_word   : bool;

	expected_ret_bool   : bool;
	expected_ret_byte   : bool;
	expected_ret_dint   : bool;
	expected_ret_dword  : bool;
	expected_ret_int    : bool;
	expected_ret_lreal  : bool;
	expected_ret_real   : bool;
	expected_ret_string : bool;
	expected_ret_time   : bool;
	expected_ret_uint   : bool;
	expected_ret_udint  : bool;
	expected_ret_word   : bool;

	index : int := 1;
	expected: string;
	obtained: string;
	result : bool;
END_VAR

	if Status = STATUS_RUNNING AND test_level_39 > TEST_DISABLED and test_loops_39 < Target then

		(* ---------- test action ---------------*)
        ret_bool   := le( lreal_to_bool(test_case[index].input0),
						 lreal_to_bool(test_case[index].input1));
        ret_byte   := le( lreal_to_byte(test_case[index].input0),
						 lreal_to_byte(test_case[index].input1));
        ret_dint   := le( lreal_to_dint(test_case[index].input0),
						 lreal_to_dint(test_case[index].input1));
        ret_dword  := le( lreal_to_dword(test_case[index].input0),
						 lreal_to_dword(test_case[index].input1));
        ret_int    := le( lreal_to_int(test_case[index].input0),
						 lreal_to_int(test_case[index].input1));
        ret_lreal  := le( test_case[index].input0,
						 test_case[index].input1);
        ret_real   := le( lreal_to_real(test_case[index].input0),
						 lreal_to_real(test_case[index].input1));
        ret_string := le(lreal_to_string(test_case[index].input0),
						 lreal_to_string(test_case[index].input1));
        ret_time   := le( lreal_to_time(test_case[index].input0),
						 lreal_to_time(test_case[index].input1));
        ret_uint   := le( lreal_to_uint(test_case[index].input0),
						 lreal_to_uint(test_case[index].input1));
        ret_udint  := le(lreal_to_udint(test_case[index].input0),
						 lreal_to_udint(test_case[index].input1));
        ret_word   := le( lreal_to_word(test_case[index].input0),
						 lreal_to_word(test_case[index].input1));

		IF (test_case[index].input0 <> 0.0 and test_case[index].input1 <> 0.0)
			or (test_case[index].input0 = 0.0 and test_case[index].input1 = 0.0)THEN
        	expected_ret_bool   := true;
        ELSE
        	expected_ret_bool   := false;
		END_IF;
		expected_ret_byte   := test_case[index].retval;
		expected_ret_dint   := test_case[index].retval;
		expected_ret_dword  := test_case[index].retval;
		expected_ret_int    := test_case[index].retval;
		expected_ret_lreal  := test_case[index].retval;
		expected_ret_real   := test_case[index].retval;
		expected_ret_string := test_case[index].retval;
		expected_ret_time   := test_case[index].retval;
		expected_ret_uint   := test_case[index].retval;
		expected_ret_udint  := test_case[index].retval;
		expected_ret_word   := test_case[index].retval;

		(* ---------- test condition ---------------*)
        result := (ret_bool = expected_ret_bool)
				  and (ret_byte = expected_ret_byte)
				  and (ret_dint = expected_ret_dint)
				  and (ret_dword = expected_ret_dword)
				  and (ret_int = expected_ret_int)
				  and (ret_lreal = expected_ret_lreal)
				  and (ret_real = expected_ret_real)
				  and (ret_string = expected_ret_string)
				  and (ret_time = expected_ret_time)
				  and (ret_uint = expected_ret_uint)
				  and (ret_udint = expected_ret_udint)
				  and (ret_word = expected_ret_word);

		(* ---------- log message ---------------*)
		expected := '';
		expected := CONCAT(expected, comma_blank, bool_to_string(expected_ret_bool));
		expected := CONCAT(expected, comma_blank, bool_to_string(expected_ret_byte));
		expected := CONCAT(expected, comma_blank, bool_to_string(expected_ret_dint));
		expected := CONCAT(expected, comma_blank, bool_to_string(expected_ret_dword));
		expected := CONCAT(expected, comma_blank, bool_to_string(expected_ret_int));
		expected := CONCAT(expected, comma_blank, bool_to_string(expected_ret_lreal));
		expected := CONCAT(expected, comma_blank, bool_to_string(expected_ret_real));
		expected := CONCAT(expected, comma_blank, bool_to_string(expected_ret_string));
		expected := CONCAT(expected, comma_blank, bool_to_string(expected_ret_time));
		expected := CONCAT(expected, comma_blank, bool_to_string(expected_ret_uint));
		expected := CONCAT(expected, comma_blank, bool_to_string(expected_ret_udint));
		expected := CONCAT(expected, comma_blank, bool_to_string(expected_ret_word));

		obtained := '';
		obtained := CONCAT(obtained, comma_blank, bool_to_string(ret_bool));
		obtained := CONCAT(obtained, comma_blank, bool_to_string(ret_byte));
		obtained := CONCAT(obtained, comma_blank, bool_to_string(ret_dint));
		obtained := CONCAT(obtained, comma_blank, bool_to_string(ret_dword));
		obtained := CONCAT(obtained, comma_blank, bool_to_string(ret_int));
		obtained := CONCAT(obtained, comma_blank, bool_to_string(ret_lreal));
		obtained := CONCAT(obtained, comma_blank, bool_to_string(ret_real));
		obtained := CONCAT(obtained, comma_blank, bool_to_string(ret_string));
		obtained := CONCAT(obtained, comma_blank, bool_to_string(ret_time));
		obtained := CONCAT(obtained, comma_blank, bool_to_string(ret_uint));
		obtained := CONCAT(obtained, comma_blank, bool_to_string(ret_udint));
		obtained := CONCAT(obtained, comma_blank, bool_to_string(ret_word));

		(* ---------- cycle ----------*)
		SingleTest(this, result, expected, obtained, test_cases,
				   index, test_level_39, test_counter_39, test_loops_39, test_errors_39);
	end_if;

END_PROGRAM

(* ---- left_right_P.st ---- *)
(*[[ ]]*)
PROGRAM left_right_P
#import "Crosstable.gvl"
#import "Resource1.gvl"
CONST
	this : int := 46;
	test_cases : int := 3;
END_CONST
VAR
	test_case : array [1..test_cases] of string_int_string2_T := [
		(input0 := 'stringa_di_partenza', input1 := 0, retval0 := '', retval1 := ''),
		(input0 := 'stringa_di_partenza', input1 := 2, retval0 := 'st', retval1 := 'za'),
		(input0 := 'stringa_di_partenza', input1 := 7, retval0 := 'stringa', retval1 := 'artenza')
	];
    retval0   : string;
    retval1   : string;
    retval2   : string;
    retval3   : string;

	index : int := 1;
	expected : string;
	obtained : string;
	result : bool;
END_VAR

	if Status = STATUS_RUNNING AND test_level_46 > TEST_DISABLED and test_loops_46 < Target then

		(* ---------- test action ---------------*)
        retval0 := left(test_case[index].input0, test_case[index].input1);
        retval1 := left(test_case[index].input0, int_to_dint(test_case[index].input1));
        retval2 := right(test_case[index].input0, test_case[index].input1);
        retval3 := right(test_case[index].input0, int_to_dint(test_case[index].input1));

		(* ---------- test condition ---------------*)
        result := (retval0 = test_case[index].retval0)
		      and (retval1 = test_case[index].retval0)
		      and (retval2 = test_case[index].retval1)
		      and (retval3 = test_case[index].retval1);

		(* ---------- log message ---------------*)
		expected := '';
		expected := CONCAT(expected, comma_blank, test_case[index].retval0);
		expected := CONCAT(expected, comma_blank, test_case[index].retval0);
		expected := CONCAT(expected, comma_blank, test_case[index].retval1);
		expected := CONCAT(expected, comma_blank, test_case[index].retval1);
		obtained := '';
		obtained := CONCAT(obtained, comma_blank, retval0);
		obtained := CONCAT(obtained, comma_blank, retval1);
		obtained := CONCAT(obtained, comma_blank, retval2);
		obtained := CONCAT(obtained, comma_blank, retval3);

		(* ---------- cycle ----------*)
		SingleTest(this, result, expected, obtained, test_cases,
				   index, test_level_46, test_counter_46, test_loops_46, test_errors_46);
	end_if;
END_PROGRAM

(* ---- len_P.st ---- *)
(*[[ ]]*)
PROGRAM len_P
#import "Crosstable.gvl"
#import "Resource1.gvl"
CONST
	this : int := 47;
	test_cases : int := 3;
END_CONST
VAR
	test_case : array [1..test_cases] of string_int_T := [
		(input := '', retval := 0),
		(input := 'stringa_in_cui_eseguire_la_ricerca', retval := 34),
		(input := 'Buzz, Woody e Jessie', retval := 20)
	];
    retval0   : int;
    retval1   : dint;

	index : int := 1;
	expected : string;
	obtained : string;
	result : bool;
END_VAR

	if Status = STATUS_RUNNING AND test_level_47 > TEST_DISABLED and test_loops_47 < Target then

		(* ---------- test action ---------------*)
        retval0 := len(test_case[index].input);
        retval1 := len(test_case[index].input);

		(* ---------- test condition ---------------*)
        result := (retval0 = test_case[index].retval)
		      and (retval1 = int_to_dint(test_case[index].retval));

		(* ---------- log message ---------------*)
		expected := '';
		expected := CONCAT(expected, comma_blank, int_to_string(test_case[index].retval));
		expected := CONCAT(expected, comma_blank, int_to_string(test_case[index].retval));
		obtained := '';
		obtained := CONCAT(obtained, comma_blank, int_to_string(retval0));
		obtained := CONCAT(obtained, comma_blank, dint_to_string(retval1));

		(* ---------- cycle ----------*)
		SingleTest(this, result, expected, obtained, test_cases,
				   index, test_level_47, test_counter_47, test_loops_47, test_errors_47);
	end_if;
END_PROGRAM

(* ---- limit_P.st ---- *)
(*[[ ]]*)
PROGRAM limit_P
#import "Crosstable.gvl"
#import "Resource1.gvl"
CONST
	this : int := 31;
	test_cases : int := 4;
END_CONST
VAR
	test_case : array [1..test_cases] of num3_num_T := [
		(input0 := 10.0,  input1 := 20.0,  input2 := 30.0,  ret_byte := 20, ret_word := 20, ret_dword := 20, ret_int := 20, ret_dint := 20,
															ret_time := t#20ms, ret_real := 20.0, ret_lreal := 20.0, ret_string := '20'),
		(input0 := 20.0,  input1 := 10.0,  input2 := 30.0,  ret_byte := 20, ret_word := 20, ret_dword := 20, ret_int := 20, ret_dint := 20,
															ret_time := t#20ms, ret_real := 20.0, ret_lreal := 20.0, ret_string := '20'),
		(input0 := 10.0,  input1 := 90.0, input2 := 20.0,  ret_byte := 20, ret_word := 20, ret_dword := 20, ret_int := 20, ret_dint := 20,
															ret_time := t#20ms, ret_real := 20.0, ret_lreal := 20.0, ret_string := '20'),
		(input0 := 20.0,  input1 := 90.0, input2 := 20.0,  ret_byte := 20, ret_word := 20, ret_dword := 20, ret_int := 20, ret_dint := 20,
															ret_time := t#20ms, ret_real := 20.0, ret_lreal := 20.0, ret_string := '20')
	];
    ret_byte   : byte;
    ret_word   : word;
    ret_dword  : dword;
    ret_int    : int;
    ret_dint   : dint;
    ret_time   : time;
    ret_real   : real;
    ret_lreal  : lreal;
    ret_string : string;

	index : int := 1;
	expected : string;
	obtained : string;
	result : bool;
END_VAR

	if Status = STATUS_RUNNING AND test_level_31 > TEST_DISABLED and test_loops_31 < Target then

		(* ---------- test action ---------------*)
        ret_byte    := limit(lreal_to_byte(test_case[index].input0), lreal_to_byte(test_case[index].input1), lreal_to_byte(test_case[index].input2));
        ret_word    := limit(lreal_to_word(test_case[index].input0), lreal_to_word(test_case[index].input1), lreal_to_word(test_case[index].input2));
        ret_dword   := limit(lreal_to_dword(test_case[index].input0), lreal_to_dword(test_case[index].input1), lreal_to_dword(test_case[index].input2));
        ret_int     := limit(lreal_to_int(test_case[index].input0), lreal_to_int(test_case[index].input1), lreal_to_int(test_case[index].input2));
        ret_dint    := limit(lreal_to_dint(test_case[index].input0), lreal_to_dint(test_case[index].input1), lreal_to_dint(test_case[index].input2));
        ret_time    := limit(lreal_to_time(test_case[index].input0), lreal_to_time(test_case[index].input1), lreal_to_time(test_case[index].input2));
        ret_real    := limit(lreal_to_real(test_case[index].input0), lreal_to_real(test_case[index].input1), lreal_to_real(test_case[index].input2));
        ret_lreal   := limit(test_case[index].input0, test_case[index].input1, test_case[index].input2);
        ret_string    := limit(lreal_to_string(test_case[index].input0), lreal_to_string(test_case[index].input1), lreal_to_string(test_case[index].input2));

		(* ---------- test condition ---------------*)
        result := ((ret_byte = test_case[index].ret_byte)
			  and (ret_word = test_case[index].ret_word)
			  and (ret_dword = test_case[index].ret_dword)
			  and (ret_int = test_case[index].ret_int)
		      and (ret_dint = test_case[index].ret_dint)
		      and (ret_time = test_case[index].ret_time)
		      and (ret_real = test_case[index].ret_real)
		      and (ret_lreal = test_case[index].ret_lreal)
		      and (ret_string = test_case[index].ret_string));

		(* ---------- log message ---------------*)
		expected := '';
		expected := CONCAT(expected, comma_blank, byte_to_string(test_case[index].ret_byte));
		expected := CONCAT(expected, comma_blank, word_to_string(test_case[index].ret_word));
		expected := CONCAT(expected, comma_blank, dword_to_string(test_case[index].ret_dword));
		expected := CONCAT(expected, comma_blank, int_to_string(test_case[index].ret_int));
		expected := CONCAT(expected, comma_blank, dint_to_string(test_case[index].ret_dint));
		expected := CONCAT(expected, comma_blank, time_to_string(test_case[index].ret_time));
		expected := CONCAT(expected, comma_blank, real_to_string(test_case[index].ret_real));
		expected := CONCAT(expected, comma_blank, lreal_to_string(test_case[index].ret_lreal));
		expected := CONCAT(expected, comma_blank, test_case[index].ret_string);
		obtained := '';
		obtained := CONCAT(obtained, comma_blank, byte_to_string(ret_byte));
		obtained := CONCAT(obtained, comma_blank, word_to_string(ret_word));
		obtained := CONCAT(obtained, comma_blank, dword_to_string(ret_dword));
		obtained := CONCAT(obtained, comma_blank, int_to_string(ret_int));
		obtained := CONCAT(obtained, comma_blank, dint_to_string(ret_dint));
		obtained := CONCAT(obtained, comma_blank, time_to_string(ret_time));
		obtained := CONCAT(obtained, comma_blank, real_to_string(ret_real));
		obtained := CONCAT(obtained, comma_blank, lreal_to_string(ret_lreal));
		obtained := CONCAT(obtained, comma_blank, ret_string);

		(* ---------- cycle ----------*)
		SingleTest(this, result, expected, obtained, test_cases,
				   index, test_level_31, test_counter_31, test_loops_31, test_errors_31);
	end_if;
END_PROGRAM

(* ---- lreal_to_all_P.st ---- *)
(*[[
]]*)
PROGRAM lreal_to_all_P
#import "Crosstable.gvl"
#import "Resource1.gvl"
CONST
	this : int := 6;
	test_cases : int := 5;
END_CONST
VAR
	test_case : array [1..test_cases] of lreal_all_T := [
		(input := 0.0, ret_bool := 0, ret_byte := 0, ret_dword := 0, ret_int := 0, ret_dint := 0, ret_real := 0.0,
		   ret_string := '0', ret_time := t#0ms, ret_udint := 0, ret_uint := 0, ret_word := 0),
		(input := 1.0, ret_bool := 1, ret_byte := 1, ret_dword := 1, ret_int := 1, ret_dint := 1, ret_real := 1.0,
		   ret_string := '1', ret_time := t#1ms, ret_udint := 1, ret_uint := 1, ret_word := 1),
		(input := -1.0, ret_bool := 1, ret_byte := 0, ret_dword := 0, ret_int := -1, ret_dint := -1, ret_real := -1.0,
		   ret_string := '-1', ret_time := t#-1ms, ret_udint := 0, ret_uint := 0, ret_word := 0),
		(input := 255.0, ret_bool := 1, ret_byte := 255, ret_dword := 255, ret_int := 255, ret_dint := 255, ret_real := 255.0,
		   ret_string := '255', ret_time := t#255ms, ret_udint := 255, ret_uint := 255, ret_word := 255),
		(input := 400.0, ret_bool := 1, ret_byte := 255, ret_dword := 400, ret_int := 400, ret_dint := 400, ret_real := 400.0,
		   ret_string := '400', ret_time := t#400ms, ret_udint := 400, ret_uint := 400, ret_word := 400)
	];
    ret_bool   : bool;
    ret_byte   : byte;
    ret_dword  : dword;
    ret_int    : int;
    ret_dint   : dint;
    ret_real   : real;
    ret_time   : time;
    ret_string : string;
    ret_udint  : udint;
    ret_uint   : uint;
    ret_word   : word;

	index : int := 1;
	expected : string;
	obtained : string;
	result : bool;
END_VAR

	if Status = STATUS_RUNNING AND test_level_06 > TEST_DISABLED and test_loops_06 < Target then

		(* ---------- test action ---------------*)
        ret_bool   := lreal_to_bool(test_case[index].input);
        ret_byte   := lreal_to_byte(test_case[index].input);
        ret_dword  := lreal_to_dword(test_case[index].input);
        ret_int    := lreal_to_int(test_case[index].input);
        ret_dint   := lreal_to_dint(test_case[index].input);
        ret_real   := lreal_to_real(test_case[index].input);
        ret_string := lreal_to_string(test_case[index].input);
        ret_time   := lreal_to_time(test_case[index].input);
        ret_udint  := lreal_to_udint(test_case[index].input);
        ret_uint   := lreal_to_uint(test_case[index].input);
        ret_word   := lreal_to_word(test_case[index].input);

		(* ---------- test condition ---------------*)
        result := (ret_bool = test_case[index].ret_bool)
		      and (ret_byte = test_case[index].ret_byte)
		      and (ret_dword = test_case[index].ret_dword)
		      and (ret_int = test_case[index].ret_int)
		      and (ret_dint = test_case[index].ret_dint)
		      and (ret_real = test_case[index].ret_real)
		      and (ret_string = test_case[index].ret_string)
		      and (ret_time = test_case[index].ret_time)
		      and (ret_udint = test_case[index].ret_udint)
		      and (ret_uint = test_case[index].ret_uint)
		      and (ret_word = test_case[index].ret_word);

		(* ---------- log message ---------------*)
		expected := '';
		expected := CONCAT(expected, comma_blank, bool_to_string(test_case[index].ret_bool));
		expected := CONCAT(expected, comma_blank, byte_to_string(test_case[index].ret_byte));
		expected := CONCAT(expected, comma_blank, dword_to_string(test_case[index].ret_dword));
		expected := CONCAT(expected, comma_blank, int_to_string(test_case[index].ret_int));
		expected := CONCAT(expected, comma_blank, dint_to_string(test_case[index].ret_dint));
		expected := CONCAT(expected, comma_blank, real_to_string(test_case[index].ret_real));
		expected := CONCAT(expected, comma_blank, test_case[index].ret_string);
		expected := CONCAT(expected, comma_blank, udint_to_string(test_case[index].ret_udint));
		expected := CONCAT(expected, comma_blank, time_to_string(test_case[index].ret_time));
		expected := CONCAT(expected, comma_blank, uint_to_string(test_case[index].ret_uint));
		expected := CONCAT(expected, comma_blank, word_to_string(test_case[index].ret_word));
		obtained := '';
		obtained := CONCAT(obtained, comma_blank, bool_to_string(ret_bool));
		obtained := CONCAT(obtained, comma_blank, byte_to_string(ret_byte));
		obtained := CONCAT(obtained, comma_blank, dword_to_string(ret_dword));
		obtained := CONCAT(obtained, comma_blank, int_to_string(ret_int));
		obtained := CONCAT(obtained, comma_blank, dint_to_string(ret_dint));
		obtained := CONCAT(obtained, comma_blank, real_to_string(ret_real));
		obtained := CONCAT(obtained, comma_blank, ret_string);
		obtained := CONCAT(obtained, comma_blank, time_to_string(ret_time));
		obtained := CONCAT(obtained, comma_blank, udint_to_string(ret_udint));
		obtained := CONCAT(obtained, comma_blank, uint_to_string(ret_uint));
		obtained := CONCAT(obtained, comma_blank, word_to_string(ret_word));

		(* ---------- cycle ----------*)
		SingleTest(this, result, expected, obtained, test_cases,
				   index, test_level_06, test_counter_06, test_loops_06, test_errors_06);
	end_if;

END_PROGRAM

(* ---- lt_P.st ---- *)
(*[[
]]*)
PROGRAM lt_P
#import "Crosstable.gvl"
#import "Resource1.gvl"
CONST
	this : int := 40;
	test_cases : int := 4;
END_CONST
VAR
	test_case : array [1..test_cases] of any2_bool_T := [
		(input0 :=  10.0, input1 :=  10.0, retval := false),
		(input0 :=  10.0, input1 :=  20.0, retval := true),
		(input0 :=  20.0, input1 :=  10.0,  retval := false),
		(input0 :=  -100.0, input1 := -100.0,  retval := false)
	];
	ret_bool   : bool;
	ret_byte   : bool;
	ret_dint   : bool;
	ret_dword  : bool;
	ret_int    : bool;
	ret_lreal  : bool;
	ret_real   : bool;
	ret_string : bool;
	ret_time   : bool;
	ret_uint   : bool;
	ret_udint  : bool;
	ret_word   : bool;

	expected_ret_bool   : bool;
	expected_ret_byte   : bool;
	expected_ret_dint   : bool;
	expected_ret_dword  : bool;
	expected_ret_int    : bool;
	expected_ret_lreal  : bool;
	expected_ret_real   : bool;
	expected_ret_string : bool;
	expected_ret_time   : bool;
	expected_ret_uint   : bool;
	expected_ret_udint  : bool;
	expected_ret_word   : bool;

	index : int := 1;
	expected: string;
	obtained: string;
	result : bool;
END_VAR

	if Status = STATUS_RUNNING AND test_level_40 > TEST_DISABLED and test_loops_40 < Target then

		(* ---------- test action ---------------*)
        ret_bool   := lt( lreal_to_bool(test_case[index].input0),
						 lreal_to_bool(test_case[index].input1));
        ret_byte   := lt( lreal_to_byte(test_case[index].input0),
						 lreal_to_byte(test_case[index].input1));
        ret_dint   := lt( lreal_to_dint(test_case[index].input0),
						 lreal_to_dint(test_case[index].input1));
        ret_dword  := lt( lreal_to_dword(test_case[index].input0),
						 lreal_to_dword(test_case[index].input1));
        ret_int    := lt( lreal_to_int(test_case[index].input0),
						 lreal_to_int(test_case[index].input1));
        ret_lreal  := lt( test_case[index].input0,
						 test_case[index].input1);
        ret_real   := lt( lreal_to_real(test_case[index].input0),
						 lreal_to_real(test_case[index].input1));
        ret_string := lt(lreal_to_string(test_case[index].input0),
						 lreal_to_string(test_case[index].input1));
        ret_time   := lt( lreal_to_time(test_case[index].input0),
						 lreal_to_time(test_case[index].input1));
        ret_uint   := lt( lreal_to_uint(test_case[index].input0),
						 lreal_to_uint(test_case[index].input1));
        ret_udint  := lt(lreal_to_udint(test_case[index].input0),
						 lreal_to_udint(test_case[index].input1));
        ret_word   := lt( lreal_to_word(test_case[index].input0),
						 lreal_to_word(test_case[index].input1));

		IF (test_case[index].input0 <> 0.0 and test_case[index].input1 <> 0.0)
			or (test_case[index].input0 = 0.0 and test_case[index].input1 = 0.0)THEN
        	expected_ret_bool   := false;
        ELSE
        	expected_ret_bool   := true;
		END_IF;
		expected_ret_byte   := test_case[index].retval;
		expected_ret_dint   := test_case[index].retval;
		expected_ret_dword  := test_case[index].retval;
		expected_ret_int    := test_case[index].retval;
		expected_ret_lreal  := test_case[index].retval;
		expected_ret_real   := test_case[index].retval;
		expected_ret_string := test_case[index].retval;
		expected_ret_time   := test_case[index].retval;
		expected_ret_uint   := test_case[index].retval;
		expected_ret_udint  := test_case[index].retval;
		expected_ret_word   := test_case[index].retval;

		(* ---------- test condition ---------------*)
        result := (ret_bool = expected_ret_bool)
				  and (ret_byte = expected_ret_byte)
				  and (ret_dint = expected_ret_dint)
				  and (ret_dword = expected_ret_dword)
				  and (ret_int = expected_ret_int)
				  and (ret_lreal = expected_ret_lreal)
				  and (ret_real = expected_ret_real)
				  and (ret_string = expected_ret_string)
				  and (ret_time = expected_ret_time)
				  and (ret_uint = expected_ret_uint)
				  and (ret_udint = expected_ret_udint)
				  and (ret_word = expected_ret_word);

		(* ---------- log message ---------------*)
		expected := '';
		expected := CONCAT(expected, comma_blank, bool_to_string(expected_ret_bool));
		expected := CONCAT(expected, comma_blank, bool_to_string(expected_ret_byte));
		expected := CONCAT(expected, comma_blank, bool_to_string(expected_ret_dint));
		expected := CONCAT(expected, comma_blank, bool_to_string(expected_ret_dword));
		expected := CONCAT(expected, comma_blank, bool_to_string(expected_ret_int));
		expected := CONCAT(expected, comma_blank, bool_to_string(expected_ret_lreal));
		expected := CONCAT(expected, comma_blank, bool_to_string(expected_ret_real));
		expected := CONCAT(expected, comma_blank, bool_to_string(expected_ret_string));
		expected := CONCAT(expected, comma_blank, bool_to_string(expected_ret_time));
		expected := CONCAT(expected, comma_blank, bool_to_string(expected_ret_uint));
		expected := CONCAT(expected, comma_blank, bool_to_string(expected_ret_udint));
		expected := CONCAT(expected, comma_blank, bool_to_string(expected_ret_word));

		obtained := '';
		obtained := CONCAT(obtained, comma_blank, bool_to_string(ret_bool));
		obtained := CONCAT(obtained, comma_blank, bool_to_string(ret_byte));
		obtained := CONCAT(obtained, comma_blank, bool_to_string(ret_dint));
		obtained := CONCAT(obtained, comma_blank, bool_to_string(ret_dword));
		obtained := CONCAT(obtained, comma_blank, bool_to_string(ret_int));
		obtained := CONCAT(obtained, comma_blank, bool_to_string(ret_lreal));
		obtained := CONCAT(obtained, comma_blank, bool_to_string(ret_real));
		obtained := CONCAT(obtained, comma_blank, bool_to_string(ret_string));
		obtained := CONCAT(obtained, comma_blank, bool_to_string(ret_time));
		obtained := CONCAT(obtained, comma_blank, bool_to_string(ret_uint));
		obtained := CONCAT(obtained, comma_blank, bool_to_string(ret_udint));
		obtained := CONCAT(obtained, comma_blank, bool_to_string(ret_word));

		(* ---------- cycle ----------*)
		SingleTest(this, result, expected, obtained, test_cases,
				   index, test_level_40, test_counter_40, test_loops_40, test_errors_40);
	end_if;

END_PROGRAM

(* ---- make_word_P.st ---- *)
(*[[ ]]*)
PROGRAM make_word_P
#import "Crosstable.gvl"
#import "Resource1.gvl"
CONST
	this : int := 59;
	test_cases : int := 4;
END_CONST
VAR
	test_case : array [1..test_cases] of bit2_bit_T := [
		(input0 := 16#0000, input1 := 16#0000, ret_word := 16#0000, ret_dword := 16#00000000),
		(input0 := 16#00ff, input1 := 16#00ff, ret_word := 16#ffff, ret_dword := 16#00ff00ff),
		(input0 := 16#1234, input1 := 16#abcd, ret_word := 16#cd34, ret_dword := 16#abcd1234),
		(input0 := 16#1122, input1 := 16#3344, ret_word := 16#4422, ret_dword := 16#33441122)
	];
    ret_word   : word;
    ret_dword  : dword;

	index : int := 1;
	expected : string;
	obtained : string;
	result : bool;
END_VAR

	if Status = STATUS_RUNNING AND test_level_59 > TEST_DISABLED and test_loops_59 < Target then

		(* ---------- test action ---------------*)
        ret_dword := make_dword(dword_to_word(test_case[index].input0), dword_to_word(test_case[index].input1));
        ret_word  := make_word( dword_to_byte(test_case[index].input0), dword_to_byte(test_case[index].input1));

		(* ---------- test condition ---------------*)
        result := (ret_word = test_case[index].ret_word)
		      and (ret_dword = test_case[index].ret_dword);

		(* ---------- log message ---------------*)
		expected := '';
		expected := CONCAT(expected, comma_blank, word_to_string(test_case[index].ret_word));
		expected := CONCAT(expected, comma_blank, dword_to_string(test_case[index].ret_dword));
		obtained := '';
		obtained := CONCAT(obtained, comma_blank, word_to_string(ret_word));
		obtained := CONCAT(obtained, comma_blank, dword_to_string(ret_dword));

		(* ---------- cycle ----------*)
		SingleTest(this, result, expected, obtained, test_cases,
				   index, test_level_59, test_counter_59, test_loops_59, test_errors_59);
	end_if;
END_PROGRAM

(* ---- max_P.st ---- *)
(*[[ ]]*)
PROGRAM max_P
#import "Crosstable.gvl"
#import "Resource1.gvl"
CONST
	this : int := 32;
	test_cases : int := 3;
END_CONST
VAR
	test_case : array [1..test_cases] of any2_any_T := [
		(input0 := 10.0,  input1 := 20.0, ret_byte := 20, ret_word := 20, ret_dword := 20, ret_int := 20, ret_dint := 20,
										ret_time := t#20ms, ret_real := 20.0, ret_lreal := 20.0, ret_string := '20'),
		(input0 := 20.0,  input1 := 10.0, ret_byte := 20, ret_word := 20, ret_dword := 20, ret_int := 20, ret_dint := 20,
										ret_time := t#20ms, ret_real := 20.0, ret_lreal := 20.0, ret_string := '20'),
		(input0 := -20.0,  input1 := -30.0, ret_byte := 0, ret_word := 0, ret_dword := 0, ret_int := -20, ret_dint := -20,
										ret_time := t#-20ms, ret_real := -20.0, ret_lreal := -20.0, ret_string := '-30')
	];
    ret_byte   : byte;
    ret_word   : word;
    ret_dword  : dword;
    ret_int    : int;
    ret_dint   : dint;
    ret_time   : time;
    ret_real   : real;
    ret_lreal  : lreal;
    ret_string : string;

	index : int := 1;
	expected : string;
	obtained : string;
	result : bool;
END_VAR

	if Status = STATUS_RUNNING AND test_level_32 > TEST_DISABLED and test_loops_32 < Target then

		(* ---------- test action ---------------*)
        ret_byte    := max(lreal_to_byte(test_case[index].input0), lreal_to_byte(test_case[index].input1));
        ret_word    := max(lreal_to_word(test_case[index].input0), lreal_to_word(test_case[index].input1));
        ret_dword   := max(lreal_to_dword(test_case[index].input0), lreal_to_dword(test_case[index].input1));
        ret_int     := max(lreal_to_int(test_case[index].input0), lreal_to_int(test_case[index].input1));
        ret_dint    := max(lreal_to_dint(test_case[index].input0), lreal_to_dint(test_case[index].input1));
        ret_time    := max(lreal_to_time(test_case[index].input0), lreal_to_time(test_case[index].input1));
        ret_real    := max(lreal_to_real(test_case[index].input0), lreal_to_real(test_case[index].input1));
        ret_lreal   := max(test_case[index].input0, test_case[index].input1);
        ret_string  := max(lreal_to_string(test_case[index].input0), lreal_to_string(test_case[index].input1));

		(* ---------- test condition ---------------*)
        result := ((ret_byte = test_case[index].ret_byte)
			  and (ret_word = test_case[index].ret_word)
			  and (ret_dword = test_case[index].ret_dword)
			  and (ret_int = test_case[index].ret_int)
		      and (ret_dint = test_case[index].ret_dint)
		      and (ret_time = test_case[index].ret_time)
		      and (ret_real = test_case[index].ret_real)
		      and (ret_lreal = test_case[index].ret_lreal)
		      and (ret_string = test_case[index].ret_string));

		(* ---------- log message ---------------*)
		expected := '';
		expected := CONCAT(expected, comma_blank, byte_to_string(test_case[index].ret_byte));
		expected := CONCAT(expected, comma_blank, word_to_string(test_case[index].ret_word));
		expected := CONCAT(expected, comma_blank, dword_to_string(test_case[index].ret_dword));
		expected := CONCAT(expected, comma_blank, int_to_string(test_case[index].ret_int));
		expected := CONCAT(expected, comma_blank, dint_to_string(test_case[index].ret_dint));
		expected := CONCAT(expected, comma_blank, time_to_string(test_case[index].ret_time));
		expected := CONCAT(expected, comma_blank, real_to_string(test_case[index].ret_real));
		expected := CONCAT(expected, comma_blank, lreal_to_string(test_case[index].ret_lreal));
		expected := CONCAT(expected, comma_blank, test_case[index].ret_string);
		obtained := '';
		obtained := CONCAT(obtained, comma_blank, byte_to_string(ret_byte));
		obtained := CONCAT(obtained, comma_blank, word_to_string(ret_word));
		obtained := CONCAT(obtained, comma_blank, dword_to_string(ret_dword));
		obtained := CONCAT(obtained, comma_blank, int_to_string(ret_int));
		obtained := CONCAT(obtained, comma_blank, dint_to_string(ret_dint));
		obtained := CONCAT(obtained, comma_blank, time_to_string(ret_time));
		obtained := CONCAT(obtained, comma_blank, real_to_string(ret_real));
		obtained := CONCAT(obtained, comma_blank, lreal_to_string(ret_lreal));
		obtained := CONCAT(obtained, comma_blank, ret_string);

		(* ---------- cycle ----------*)
		SingleTest(this, result, expected, obtained, test_cases,
				   index, test_level_32, test_counter_32, test_loops_32, test_errors_32);
	end_if;
END_PROGRAM

(* ---- mid_P.st ---- *)
(*[[ ]]*)
PROGRAM mid_P
#import "Crosstable.gvl"
#import "Resource1.gvl"
CONST
	this : int := 48;
	test_cases : int := 4;
END_CONST
VAR
	test_case : array [1..test_cases] of string_int2_string_T := [
		(input0 := 'stringa_di_test', input1 := 3,   input2 := 8, retval := '_di'),
		(input0 := 'stringa_di_test', input1 := 11,  input2 := 0, retval := 'stringa_di_'),
		(input0 := 'stringa_di_test', input1 := 8,   input2 := 8, retval := '_di_test'),
		(input0 := 'stringa_di_test', input1 := 100, input2 := 8, retval := '_di_test')
	];
    retval0   : string;
    retval1   : string;

	index : int := 1;
	expected : string;
	obtained : string;
	result : bool;
END_VAR

	if Status = STATUS_RUNNING AND test_level_48 > TEST_DISABLED and test_loops_48 < Target then

		(* ---------- test action ---------------*)
        retval0 := mid(test_case[index].input0, test_case[index].input1, test_case[index].input2);
        retval1 := mid(test_case[index].input0, int_to_dint(test_case[index].input1), int_to_dint(test_case[index].input2));

		(* ---------- test condition ---------------*)
        result := (retval0 = test_case[index].retval)
		      and (retval1 = test_case[index].retval);

		(* ---------- log message ---------------*)
		expected := '';
		expected := CONCAT(expected, comma_blank, test_case[index].retval);
		expected := CONCAT(expected, comma_blank, test_case[index].retval);
		obtained := '';
		obtained := CONCAT(obtained, comma_blank, retval0);
		obtained := CONCAT(obtained, comma_blank, retval1);

		(* ---------- cycle ----------*)
		SingleTest(this, result, expected, obtained, test_cases,
				   index, test_level_48, test_counter_48, test_loops_48, test_errors_48);
	end_if;
END_PROGRAM

(* ---- min_P.st ---- *)
(*[[ ]]*)
PROGRAM min_P
#import "Crosstable.gvl"
#import "Resource1.gvl"
CONST
	this : int := 33;
	test_cases : int := 4;
END_CONST
VAR
	test_case : array [1..test_cases] of any2_any_T := [
		(input0 := 30.0,  input1 := 20.0, ret_byte := 20, ret_word := 20, ret_dword := 20, ret_int := 20, ret_dint := 20,
										ret_time := t#20ms, ret_real := 20.0, ret_lreal := 20.0, ret_string := '20'),
		(input0 := 20.0,  input1 := 30.0, ret_byte := 20, ret_word := 20, ret_dword := 20, ret_int := 20, ret_dint := 20,
										ret_time := t#20ms, ret_real := 20.0, ret_lreal := 20.0, ret_string := '20'),
		(input0 := 20.0,  input1 := 20.0, ret_byte := 20, ret_word := 20, ret_dword := 20, ret_int := 20, ret_dint := 20,
										ret_time := t#20ms, ret_real := 20.0, ret_lreal := 20.0, ret_string := '20'),
		(input0 := -20.0, input1 := -10.0, ret_byte := 0, ret_word := 0, ret_dword := 0, ret_int := -20, ret_dint := -20,
										ret_time := t#-20ms, ret_real := -20.0, ret_lreal := -20.0, ret_string := '-10')
	];
    ret_byte   : byte;
    ret_word   : word;
    ret_dword  : dword;
    ret_int    : int;
    ret_dint   : dint;
    ret_time   : time;
    ret_real   : real;
    ret_lreal  : lreal;
    ret_string : string;

	index : int := 1;
	expected : string;
	obtained : string;
	result : bool;
END_VAR

	if Status = STATUS_RUNNING AND test_level_33 > TEST_DISABLED and test_loops_33 < Target then
		(* ---------- test action ---------------*)
        ret_byte    := min(lreal_to_byte(test_case[index].input0), lreal_to_byte(test_case[index].input1));
        ret_word    := min(lreal_to_word(test_case[index].input0), lreal_to_word(test_case[index].input1));
        ret_dword   := min(lreal_to_dword(test_case[index].input0), lreal_to_dword(test_case[index].input1));
        ret_int     := min(lreal_to_int(test_case[index].input0), lreal_to_int(test_case[index].input1));
        ret_dint    := min(lreal_to_dint(test_case[index].input0), lreal_to_dint(test_case[index].input1));
        ret_time    := min(lreal_to_time(test_case[index].input0), lreal_to_time(test_case[index].input1));
        ret_real    := min(lreal_to_real(test_case[index].input0), lreal_to_real(test_case[index].input1));
        ret_lreal   := min(test_case[index].input0, test_case[index].input1);
        ret_string  := min(lreal_to_string(test_case[index].input0), lreal_to_string(test_case[index].input1));

		(* ---------- test condition ---------------*)
        result := ((ret_byte = test_case[index].ret_byte)
			  and (ret_word = test_case[index].ret_word)
			  and (ret_dword = test_case[index].ret_dword)
			  and (ret_int = test_case[index].ret_int)
		      and (ret_dint = test_case[index].ret_dint)
		      and (ret_time = test_case[index].ret_time)
		      and (ret_real = test_case[index].ret_real)
		      and (ret_lreal = test_case[index].ret_lreal)
		      and (ret_string = test_case[index].ret_string));

		(* ---------- log message ---------------*)
		expected := '';
		expected := CONCAT(expected, comma_blank, byte_to_string(test_case[index].ret_byte));
		expected := CONCAT(expected, comma_blank, word_to_string(test_case[index].ret_word));
		expected := CONCAT(expected, comma_blank, dword_to_string(test_case[index].ret_dword));
		expected := CONCAT(expected, comma_blank, int_to_string(test_case[index].ret_int));
		expected := CONCAT(expected, comma_blank, dint_to_string(test_case[index].ret_dint));
		expected := CONCAT(expected, comma_blank, time_to_string(test_case[index].ret_time));
		expected := CONCAT(expected, comma_blank, real_to_string(test_case[index].ret_real));
		expected := CONCAT(expected, comma_blank, lreal_to_string(test_case[index].ret_lreal));
		expected := CONCAT(expected, comma_blank, test_case[index].ret_string);
		obtained := '';
		obtained := CONCAT(obtained, comma_blank, byte_to_string(ret_byte));
		obtained := CONCAT(obtained, comma_blank, word_to_string(ret_word));
		obtained := CONCAT(obtained, comma_blank, dword_to_string(ret_dword));
		obtained := CONCAT(obtained, comma_blank, int_to_string(ret_int));
		obtained := CONCAT(obtained, comma_blank, dint_to_string(ret_dint));
		obtained := CONCAT(obtained, comma_blank, time_to_string(ret_time));
		obtained := CONCAT(obtained, comma_blank, real_to_string(ret_real));
		obtained := CONCAT(obtained, comma_blank, lreal_to_string(ret_lreal));
		obtained := CONCAT(obtained, comma_blank, ret_string);

		(* ---------- cycle ----------*)
		SingleTest(this, result, expected, obtained, test_cases,
				   index, test_level_33, test_counter_33, test_loops_33, test_errors_33);
	end_if;
END_PROGRAM

(* ---- mod_P.st ---- *)
(*[[ ]]*)
PROGRAM mod_P
#import "Crosstable.gvl"
#import "Resource1.gvl"
CONST
	this : int := 21;
	test_cases : int := 4;
END_CONST
VAR
	test_case : array [1..test_cases] of dint2_dint_int_T := [
		(input0 := 10, input1 := 10, ret_dint := 0, ret_int := 0),
		(input0 := 10, input1 :=  2, ret_dint := 0, ret_int := 0),
		(input0 := 11, input1 :=  2, ret_dint := 1, ret_int := 1),
		(input0 := 13, input1 :=  5, ret_dint := 3, ret_int := 3)
	];
    ret_int  : int;
    ret_dint : dint;

	index : int := 1;
	expected : string;
	obtained : string;
	result : bool;
END_VAR

	if Status = STATUS_RUNNING AND test_level_21 > TEST_DISABLED and test_loops_21 < Target then

		(* ---------- test action ---------------*)
        ret_dint   := mod(test_case[index].input0, test_case[index].input1);
        ret_int    := mod(dint_to_int(test_case[index].input0), dint_to_int(test_case[index].input1));

		(* ---------- test condition ---------------*)
        result := ((ret_int = test_case[index].ret_int)
		      and (ret_dint = test_case[index].ret_dint));

		(* ---------- log message ---------------*)
		expected := '';
		expected := CONCAT(expected, comma_blank, int_to_string(test_case[index].ret_int));
		expected := CONCAT(expected, comma_blank, dint_to_string(test_case[index].ret_dint));
		obtained := '';
		obtained := CONCAT(obtained, comma_blank, int_to_string(ret_int));
		obtained := CONCAT(obtained, comma_blank, dint_to_string(ret_dint));

		(* ---------- cycle ----------*)
		SingleTest(this, result, expected, obtained, test_cases,
				   index, test_level_21, test_counter_21, test_loops_21, test_errors_21);
	end_if;
END_PROGRAM

(* ---- move_P.st ---- *)
(*[[
]]*)
PROGRAM move_P
#import "Crosstable.gvl"
#import "Resource1.gvl"
CONST
	this : int := 22;
	test_cases : int := 2;
END_CONST
VAR
	test_case : array [1..test_cases] of dint_dint_T := [
		(input := 42, retval := 42),
		(input := -42, retval := -42)
	];
    ret_dint : dint;

	index : int := 1;
	expected : string;
	obtained : string;
	result : bool;
END_VAR

	if Status = STATUS_RUNNING AND test_level_22 > TEST_DISABLED and test_loops_22 < Target then

		(* ---------- test action ---------------*)
        ret_dint   := move(test_case[index].input);

		(* ---------- test condition ---------------*)
        result := (ret_dint = test_case[index].retval);

		(* ---------- log message ---------------*)
		expected := '';
		expected := CONCAT(expected, comma_blank, dint_to_string(test_case[index].retval));
		obtained := '';
		obtained := CONCAT(obtained, comma_blank, dint_to_string(ret_dint));

		(* ---------- cycle ----------*)
		SingleTest(this, result, expected, obtained, test_cases,
				   index, test_level_22, test_counter_22, test_loops_22, test_errors_22);
   end_if;
END_PROGRAM

(* ---- mul_P.st ---- *)
(*[[ ]]*)
PROGRAM mul_P
#import "Crosstable.gvl"
#import "Resource1.gvl"
CONST
	this : int := 23;
	test_cases : int := 4;
END_CONST
VAR
	test_case : array [1..test_cases] of num2_num_T := [
		(input0 := 10.0, input1 := 10.0, ret_int := 100, ret_dint := 100, ret_udint := 100, ret_uint := 100, ret_real := 100.0, ret_lreal := 100.0),
		(input0 := 10.0, input1 := 2.0, ret_int := 20, ret_dint := 20, ret_udint := 20, ret_uint := 20, ret_real := 20.0, ret_lreal := 20.0),
		(input0 := -10.0, input1 := -30.0, ret_int := 300, ret_dint := 300, ret_udint := 0, ret_uint := 0, ret_real := 300.0, ret_lreal := 300.0),
		(input0 := -10.0, input1 := 5.0, ret_int := -50, ret_dint := -50, ret_udint := 0, ret_uint := 0, ret_real := -50.0, ret_lreal := -50.0)
	];
    ret_int    : int;
    ret_dint   : dint;
    ret_uint   : uint;
    ret_udint  : udint;
    ret_real   : real;
    ret_lreal  : lreal;

	index : int := 1;
	expected : string;
	obtained : string;
	result : bool;
END_VAR

	if Status = STATUS_RUNNING AND test_level_23 > TEST_DISABLED and test_loops_23 < Target then

		(* ---------- test action ---------------*)
        ret_int     := mul(lreal_to_int(test_case[index].input0), lreal_to_int(test_case[index].input1));
        ret_dint    := mul(lreal_to_dint(test_case[index].input0), lreal_to_dint(test_case[index].input1));
        ret_uint    := mul(lreal_to_uint(test_case[index].input0), lreal_to_uint(test_case[index].input1));
        ret_udint   := mul(lreal_to_udint(test_case[index].input0), lreal_to_udint(test_case[index].input1));
        ret_real    := mul(lreal_to_real(test_case[index].input0), lreal_to_real(test_case[index].input1));
        ret_lreal   := mul(test_case[index].input0, test_case[index].input1);

		(* ---------- test condition ---------------*)
        result := ((ret_int = test_case[index].ret_int)
		      and (ret_dint = test_case[index].ret_dint)
		      and (ret_uint = test_case[index].ret_uint)
		      and (ret_udint = test_case[index].ret_udint)
		      and (ret_real = test_case[index].ret_real)
		      and (ret_lreal = test_case[index].ret_lreal));

		(* ---------- log message ---------------*)
		expected := '';
		expected := CONCAT(expected, comma_blank, int_to_string(test_case[index].ret_int));
		expected := CONCAT(expected, comma_blank, dint_to_string(test_case[index].ret_dint));
		expected := CONCAT(expected, comma_blank, uint_to_string(test_case[index].ret_uint));
		expected := CONCAT(expected, comma_blank, udint_to_string(test_case[index].ret_udint));
		expected := CONCAT(expected, comma_blank, real_to_string(test_case[index].ret_real));
		expected := CONCAT(expected, comma_blank, lreal_to_string(test_case[index].ret_lreal));
		obtained := '';
		obtained := CONCAT(obtained, comma_blank, int_to_string(ret_int));
		obtained := CONCAT(obtained, comma_blank, dint_to_string(ret_dint));
		obtained := CONCAT(obtained, comma_blank, uint_to_string(ret_uint));
		obtained := CONCAT(obtained, comma_blank, udint_to_string(ret_udint));
		obtained := CONCAT(obtained, comma_blank, real_to_string(ret_real));
		obtained := CONCAT(obtained, comma_blank, lreal_to_string(ret_lreal));

		(* ---------- cycle ----------*)
		SingleTest(this, result, expected, obtained, test_cases,
				   index, test_level_23, test_counter_23, test_loops_23, test_errors_23);
	end_if;
END_PROGRAM

(* ---- mux_P.st ---- *)
(*[[
]]*)
PROGRAM mux_P
#import "Crosstable.gvl"
#import "Resource1.gvl"
CONST
	this : int := 34;
	test_cases : int := 3;
END_CONST
VAR
	test_case : array [1..test_cases] of int_any3_any_T := [
		(input := 0, input0 :=  1.0, input1 :=  2.0, input2 :=  3.0, retval := 1.0),
		(input := 1, input0 :=  1.0, input1 :=  2.0, input2 :=  3.0, retval := 2.0),
		(input := 2, input0 :=  1.0, input1 :=  2.0, input2 :=  3.0, retval := 3.0)
	];
	ret_bool  : bool;
	ret_byte  : byte;
	ret_int   : int;
	ret_word  : word;
	ret_dint  : dint;
	ret_dword : dword;
	ret_time  : time;
	ret_real  : real;
	ret_lreal : lreal;
	ret_string : string;

	expected_ret_bool  : bool;
	expected_ret_byte  : byte;
	expected_ret_int   : int;
	expected_ret_word  : word;
	expected_ret_dint  : dint;
	expected_ret_dword : dword;
	expected_ret_time  : time;
	expected_ret_real  : real;
	expected_ret_lreal : lreal;
	expected_ret_string : string;

	index : int := 1;
	expected : string;
	obtained : string;
	result : bool;
END_VAR

	if Status = STATUS_RUNNING AND test_level_34 > TEST_DISABLED and test_loops_34 < Target then

		(* ---------- test action ---------------*)
        ret_bool  := mux(test_case[index].input,
						 lreal_to_bool(test_case[index].input0),
						 lreal_to_bool(test_case[index].input1),
						 lreal_to_bool(test_case[index].input2));
        ret_byte  := mux(test_case[index].input,
						 lreal_to_byte(test_case[index].input0),
						 lreal_to_byte(test_case[index].input1),
						 lreal_to_byte(test_case[index].input2));
        ret_int  := mux(test_case[index].input,
						 lreal_to_int(test_case[index].input0),
						 lreal_to_int(test_case[index].input1),
						 lreal_to_int(test_case[index].input2));
        ret_word  := mux(test_case[index].input,
						 lreal_to_word(test_case[index].input0),
						 lreal_to_word(test_case[index].input1),
						 lreal_to_word(test_case[index].input2));
        ret_dint  := mux(test_case[index].input,
						 lreal_to_dint(test_case[index].input0),
						 lreal_to_dint(test_case[index].input1),
						 lreal_to_dint(test_case[index].input2));
        ret_dword  := mux(test_case[index].input,
						 lreal_to_dword(test_case[index].input0),
						 lreal_to_dword(test_case[index].input1),
						 lreal_to_dword(test_case[index].input2));
        ret_time  := mux(test_case[index].input,
						 lreal_to_time(test_case[index].input0),
						 lreal_to_time(test_case[index].input1),
						 lreal_to_time(test_case[index].input2));
        ret_real  := mux(test_case[index].input,
						 lreal_to_real(test_case[index].input0),
						 lreal_to_real(test_case[index].input1),
						 lreal_to_real(test_case[index].input2));
        ret_lreal  := mux(test_case[index].input,
						 test_case[index].input0,
						 test_case[index].input1,
						 test_case[index].input2);
        ret_string  := mux(test_case[index].input,
						 lreal_to_string(test_case[index].input0),
						 lreal_to_string(test_case[index].input1),
						 lreal_to_string(test_case[index].input2));

		expected_ret_bool   := lreal_to_bool(test_case[index].retval);
		expected_ret_byte   := lreal_to_byte(test_case[index].retval);
		expected_ret_int    := lreal_to_int(test_case[index].retval);
		expected_ret_word   := lreal_to_word(test_case[index].retval);
		expected_ret_dint   := lreal_to_dint(test_case[index].retval);
		expected_ret_dword  := lreal_to_dword(test_case[index].retval);
		expected_ret_time   := lreal_to_time(test_case[index].retval);
		expected_ret_real   := lreal_to_real(test_case[index].retval);
		expected_ret_lreal  := test_case[index].retval;
		expected_ret_string := lreal_to_string(test_case[index].retval);

		(* ---------- test condition ---------------*)
        result := (ret_bool = expected_ret_bool)
				  and (ret_byte = expected_ret_byte)
				  and (ret_int = expected_ret_int)
				  and (ret_word = expected_ret_word)
				  and (ret_dint = expected_ret_dint)
				  and (ret_dword = expected_ret_dword)
				  and (ret_time = expected_ret_time)
				  and (ret_real = expected_ret_real)
				  and (ret_lreal = expected_ret_lreal)
				  and (ret_string = expected_ret_string);

		(* ---------- log message ---------------*)
		expected := '';
		expected := CONCAT(expected, comma_blank, bool_to_string(expected_ret_bool));
		expected := CONCAT(expected, comma_blank, byte_to_string(expected_ret_byte));
		expected := CONCAT(expected, comma_blank, int_to_string(expected_ret_int));
		expected := CONCAT(expected, comma_blank, word_to_string(expected_ret_word));
		expected := CONCAT(expected, comma_blank, dint_to_string(expected_ret_dint));
		expected := CONCAT(expected, comma_blank, dword_to_string(expected_ret_dword));
		expected := CONCAT(expected, comma_blank, time_to_string(expected_ret_time));
		expected := CONCAT(expected, comma_blank, real_to_string(expected_ret_real));
		expected := CONCAT(expected, comma_blank, lreal_to_string(expected_ret_lreal));
		expected := CONCAT(expected, comma_blank, expected_ret_string);
		obtained := '';
		obtained := CONCAT(obtained, comma_blank, bool_to_string(ret_bool));
		obtained := CONCAT(obtained, comma_blank, byte_to_string(ret_byte));
		obtained := CONCAT(obtained, comma_blank, int_to_string(ret_int));
		obtained := CONCAT(obtained, comma_blank, word_to_string(ret_word));
		obtained := CONCAT(obtained, comma_blank, dint_to_string(ret_dint));
		obtained := CONCAT(obtained, comma_blank, dword_to_string(ret_dword));
		obtained := CONCAT(obtained, comma_blank, time_to_string(ret_time));
		obtained := CONCAT(obtained, comma_blank, real_to_string(ret_real));
		obtained := CONCAT(obtained, comma_blank, lreal_to_string(ret_lreal));
		obtained := CONCAT(obtained, comma_blank, ret_string);

		(* ---------- cycle ----------*)
		SingleTest(this, result, expected, obtained, test_cases,
				   index, test_level_34, test_counter_34, test_loops_34, test_errors_34);
	end_if;

END_PROGRAM

(* ---- ne_P.st ---- *)
(*[[
]]*)
PROGRAM ne_P
#import "Crosstable.gvl"
#import "Resource1.gvl"
CONST
	this : int := 41;
	test_cases : int := 6;
END_CONST
VAR
	test_case : array [1..test_cases] of any2_bool_T := [
		(input0 :=  10.0, input1 :=  10.0, retval := false),
		(input0 :=  10.0, input1 :=  20.0, retval := true),
		(input0 :=  10.0, input1 :=  5.0,  retval := true),
		(input0 :=  -100.0, input1 := -100.0,  retval := false),
		(input0 :=  -100.0, input1 := 7.0,  retval := true),
		(input0 :=  -100.0, input1 := 109.0,  retval := true)
	];
	ret_bool   : bool;
	ret_byte   : bool;
	ret_dint   : bool;
	ret_dword  : bool;
	ret_int    : bool;
	ret_lreal  : bool;
	ret_real   : bool;
	ret_string : bool;
	ret_time   : bool;
	ret_uint   : bool;
	ret_udint  : bool;
	ret_word   : bool;

	expected_ret_bool   : bool;
	expected_ret_byte   : bool;
	expected_ret_dint   : bool;
	expected_ret_dword  : bool;
	expected_ret_int    : bool;
	expected_ret_lreal  : bool;
	expected_ret_real   : bool;
	expected_ret_string : bool;
	expected_ret_time   : bool;
	expected_ret_uint   : bool;
	expected_ret_udint  : bool;
	expected_ret_word   : bool;

	index : int := 1;
	expected: string;
	obtained: string;
	result : bool;
END_VAR

	if Status = STATUS_RUNNING AND test_level_41 > TEST_DISABLED and test_loops_41 < Target then

		(* ---------- test action ---------------*)
        ret_bool   := ne( lreal_to_bool(test_case[index].input0),
						 lreal_to_bool(test_case[index].input1));
        ret_byte   := ne( lreal_to_byte(test_case[index].input0),
						 lreal_to_byte(test_case[index].input1));
        ret_dint   := ne( lreal_to_dint(test_case[index].input0),
						 lreal_to_dint(test_case[index].input1));
        ret_dword  := ne( lreal_to_dword(test_case[index].input0),
						 lreal_to_dword(test_case[index].input1));
        ret_int    := ne( lreal_to_int(test_case[index].input0),
						 lreal_to_int(test_case[index].input1));
        ret_lreal  := ne( test_case[index].input0,
						 test_case[index].input1);
        ret_real   := ne( lreal_to_real(test_case[index].input0),
						 lreal_to_real(test_case[index].input1));
        ret_string := ne(lreal_to_string(test_case[index].input0),
						 lreal_to_string(test_case[index].input1));
        ret_time   := ne( lreal_to_time(test_case[index].input0),
						 lreal_to_time(test_case[index].input1));
        ret_uint   := ne( lreal_to_uint(test_case[index].input0),
						 lreal_to_uint(test_case[index].input1));
        ret_udint  := ne(lreal_to_udint(test_case[index].input0),
						 lreal_to_udint(test_case[index].input1));
        ret_word   := ne( lreal_to_word(test_case[index].input0),
						 lreal_to_word(test_case[index].input1));

		IF (test_case[index].input0 <> 0.0 and test_case[index].input1 <> 0.0)
			or (test_case[index].input0 = 0.0 and test_case[index].input1 = 0.0)THEN
        	expected_ret_bool   := false;
        ELSE
        	expected_ret_bool   := true;
		END_IF;

		expected_ret_byte   := test_case[index].retval;
		expected_ret_dint   := test_case[index].retval;
		expected_ret_dword  := test_case[index].retval;
		expected_ret_int    := test_case[index].retval;
		expected_ret_lreal  := test_case[index].retval;
		expected_ret_real   := test_case[index].retval;
		expected_ret_string := test_case[index].retval;
		expected_ret_time   := test_case[index].retval;
		expected_ret_uint   := test_case[index].retval;
		expected_ret_udint  := test_case[index].retval;
		expected_ret_word   := test_case[index].retval;

		(* ---------- test condition ---------------*)
        result := (ret_bool = expected_ret_bool)
				  and (ret_byte = expected_ret_byte)
				  and (ret_dint = expected_ret_dint)
				  and (ret_dword = expected_ret_dword)
				  and (ret_int = expected_ret_int)
				  and (ret_lreal = expected_ret_lreal)
				  and (ret_real = expected_ret_real)
				  and (ret_string = expected_ret_string)
				  and (ret_time = expected_ret_time)
				  and (ret_uint = expected_ret_uint)
				  and (ret_udint = expected_ret_udint)
				  and (ret_word = expected_ret_word);

		(* ---------- log message ---------------*)
		expected := '';
		expected := CONCAT(expected, comma_blank, bool_to_string(expected_ret_bool));
		expected := CONCAT(expected, comma_blank, bool_to_string(expected_ret_byte));
		expected := CONCAT(expected, comma_blank, bool_to_string(expected_ret_dint));
		expected := CONCAT(expected, comma_blank, bool_to_string(expected_ret_dword));
		expected := CONCAT(expected, comma_blank, bool_to_string(expected_ret_int));
		expected := CONCAT(expected, comma_blank, bool_to_string(expected_ret_lreal));
		expected := CONCAT(expected, comma_blank, bool_to_string(expected_ret_real));
		expected := CONCAT(expected, comma_blank, bool_to_string(expected_ret_string));
		expected := CONCAT(expected, comma_blank, bool_to_string(expected_ret_time));
		expected := CONCAT(expected, comma_blank, bool_to_string(expected_ret_uint));
		expected := CONCAT(expected, comma_blank, bool_to_string(expected_ret_udint));
		expected := CONCAT(expected, comma_blank, bool_to_string(expected_ret_word));

		obtained := '';
		obtained := CONCAT(obtained, comma_blank, bool_to_string(ret_bool));
		obtained := CONCAT(obtained, comma_blank, bool_to_string(ret_byte));
		obtained := CONCAT(obtained, comma_blank, bool_to_string(ret_dint));
		obtained := CONCAT(obtained, comma_blank, bool_to_string(ret_dword));
		obtained := CONCAT(obtained, comma_blank, bool_to_string(ret_int));
		obtained := CONCAT(obtained, comma_blank, bool_to_string(ret_lreal));
		obtained := CONCAT(obtained, comma_blank, bool_to_string(ret_real));
		obtained := CONCAT(obtained, comma_blank, bool_to_string(ret_string));
		obtained := CONCAT(obtained, comma_blank, bool_to_string(ret_time));
		obtained := CONCAT(obtained, comma_blank, bool_to_string(ret_uint));
		obtained := CONCAT(obtained, comma_blank, bool_to_string(ret_udint));
		obtained := CONCAT(obtained, comma_blank, bool_to_string(ret_word));

		(* ---------- cycle ----------*)
		SingleTest(this, result, expected, obtained, test_cases,
				   index, test_level_41, test_counter_41, test_loops_41, test_errors_41);
	end_if;

END_PROGRAM

(* ---- not_P.st ---- *)
(*[[ ]]*)
PROGRAM not_P
#import "Crosstable.gvl"
#import "Resource1.gvl"
CONST
	this : int := 28;
	test_cases : int := 6;
END_CONST
VAR
	test_case : array [1..test_cases] of bit2_bit_T := [
		(input0 := 1, 		    ret_bool := 0, ret_byte := 16#fe, ret_word := 16#fffe, ret_dword := 16#fffffffe),
		(input0 := 0, 		    ret_bool := 1, ret_byte := 16#ff, ret_word := 16#ffff, ret_dword := 16#ffffffff),
		(input0 := 16#000000ff, ret_bool := 0, ret_byte := 16#00, ret_word := 16#ff00, ret_dword := 16#ffffff00),
		(input0 := 16#0000000f, ret_bool := 0, ret_byte := 16#f0, ret_word := 16#fff0, ret_dword := 16#fffffff0),
		(input0 := 16#0000ffff, ret_bool := 0, ret_byte := 16#00, ret_word := 16#0000, ret_dword := 16#ffff0000),
		(input0 := 16#0000f000, ret_bool := 0, ret_byte := 16#ff, ret_word := 16#0fff, ret_dword := 16#ffff0fff)
	];
    ret_bool   : bool;
    ret_byte   : byte;
    ret_word   : word;
    ret_dword  : dword;

	index : int := 1;
	expected : string;
	obtained : string;
	result : bool;
END_VAR

	if Status = STATUS_RUNNING AND test_level_28 > TEST_DISABLED and test_loops_28 < Target then

		(* ---------- test action ---------------*)
        ret_bool   := not(dword_to_bool(test_case[index].input0));
        ret_byte   := not(dword_to_byte(test_case[index].input0));
        ret_word   := not(dword_to_word(test_case[index].input0));
        ret_dword  := not(test_case[index].input0);

		(* ---------- test condition ---------------*)
        result := (ret_bool = test_case[index].ret_bool)
		      and (ret_byte = test_case[index].ret_byte)
		      and (ret_word = test_case[index].ret_word)
		      and (ret_dword = test_case[index].ret_dword);

		(* ---------- log message ---------------*)
		expected := '';
		expected := CONCAT(expected, comma_blank, bool_to_string(test_case[index].ret_bool));
		expected := CONCAT(expected, comma_blank, byte_to_string(test_case[index].ret_byte));
		expected := CONCAT(expected, comma_blank, word_to_string(test_case[index].ret_word));
		expected := CONCAT(expected, comma_blank, dword_to_string(test_case[index].ret_dword));
		obtained := '';
		obtained := CONCAT(obtained, comma_blank, bool_to_string(ret_bool));
		obtained := CONCAT(obtained, comma_blank, byte_to_string(ret_byte));
		obtained := CONCAT(obtained, comma_blank, word_to_string(ret_word));
		obtained := CONCAT(obtained, comma_blank, dword_to_string(ret_dword));

		(* ---------- cycle ----------*)
		SingleTest(this, result, expected, obtained, test_cases,
				   index, test_level_28, test_counter_28, test_loops_28, test_errors_28);
	end_if;
END_PROGRAM
